(* Offers parameters for SB method (a simple blob detector with multiple thresholds). *)
	{attribute 'TcIecLibraryType'}
{attribute 'Namespace' := 'Tc3_Vision'}
TYPE TcVnParamsSB : 
	STRUCT
		(* Enable filtering by area (fMinArea <= area < fMaxArea). *)
		bFilterByArea : BOOL := TRUE;
		(* Enable filtering by circularity (fMinCircularity <= circularity(4pi * area / perimeter^2) < fMaxCircularity). *)
		bFilterByCircularity : BOOL := FALSE;
		(* Enable filtering by color (thresholdedColor(0 or 255) = nBlobColor). *)
		bFilterByColor : BOOL := FALSE;
		(* Enable filtering by convexity (fMinConvexity <= convexity(area / hullArea) < fMaxConvexity). *)
		bFilterByConvexity : BOOL := FALSE;
		(* Enable filtering by inertia ratio (fMinInertiaRatio <= inertia ratio < fMaxInertiaRatio). *)
		bFilterByInertia : BOOL := FALSE;
		 {attribute 'hide'}
		_reserved1 : ARRAY [1..3] OF USINT;
		(* Min estimated blob area in pixel *)
		fMinArea : REAL := 25;
		(* Max estimated blob area in pixel *)
		fMaxArea : REAL := 15000;
		(* Min circularity (1.0: ideal circle, < 1: less circular, 0: not circular at all) *)
		fMinCircularity : REAL := 0;
		(* Max circularity (1.0: ideal circle, < 1: less circular, 0: not circular at all) *)
		fMaxCircularity : REAL := 1;
		(* 0 or 255 *)
		nBlobColor : USINT := 255;
		 {attribute 'hide'}
		_reserved2 : ARRAY [1..3] OF USINT;
		(* Min convexity (1.0: blob fully convex, < 1: less convex) *)
		fMinConvexity : REAL := 0;
		(* Max convexity (1.0: blob fully convex, < 1: less convex) *)
		fMaxConvexity : REAL := 1;
		(* Min inertia ratio (0.0 .. 1.0) *)
		fMinInertiaRatio : REAL := 0;
		(* Max inertia ratio (0.0 .. 1.0) *)
		fMaxInertiaRatio : REAL := 1;
		(* Min distance between different blobs *)
		fMinBlobDist : REAL := 5;
		(* Min number of same detected blobs (dist < fMinBlobDist) in different thresholds *)
		nMinRepeatability : UDINT := 2;
		(* Min threshold (start) *)
		fMinThreshold : REAL := 30;
		(* Max threshold (stop) *)
		fMaxThreshold : REAL := 225;
		(* Threshold step between min and max threshold *)
		fThresholdStep : REAL := 10;
	END_STRUCT
END_TYPE

// TC_IID_LIST

VAR_GLOBAL
	// Interface ID for interface ITcVnCustomContainerOperation_ITcVnContainer
	{attribute 'tc_no_symbol'}
	IID_ITcVnCustomContainerOperation_ITcVnContainer: IID := (Data1 := 16#6F849123, Data2 := 16#F0E5, Data3 := 16#4EF8, Data4 := [16#99, 16#AF, 16#94, 16#C8, 16#96, 16#DC, 16#45, 16#CA]);
	// Interface ID for interface ITcVnCustomContainerOperation_ITcVnForwardIterator
	{attribute 'tc_no_symbol'}
	IID_ITcVnCustomContainerOperation_ITcVnForwardIterator: IID := (Data1 := 16#49CDB7B5, Data2 := 16#1479, Data3 := 16#4673, Data4 := [16#87, 16#51, 16#92, 16#33, 16#78, 16#F3, 16#BF, 16#4C]);
	// Interface ID for interface ITcVnCustomElementCondition_ITcVnContainer
	{attribute 'tc_no_symbol'}
	IID_ITcVnCustomElementCondition_ITcVnContainer: IID := (Data1 := 16#6B67C104, Data2 := 16#65D1, Data3 := 16#42AF, Data4 := [16#85, 16#B2, 16#AA, 16#CE, 16#B2, 16#0F, 16#60, 16#47]);
	// Interface ID for interface ITcVnCustomElementCondition_ITcVnForwardIterator
	{attribute 'tc_no_symbol'}
	IID_ITcVnCustomElementCondition_ITcVnForwardIterator: IID := (Data1 := 16#DEAD4E4B, Data2 := 16#9BBF, Data3 := 16#4E69, Data4 := [16#A4, 16#7F, 16#D5, 16#7A, 16#42, 16#C7, 16#39, 16#BC]);
	// Interface ID for interface ITcVnColorModel
	{attribute 'tc_no_symbol'}
	IID_ITcVnColorModel: IID := (Data1 := 16#0C43B589, Data2 := 16#90E8, Data3 := 16#4794, Data4 := [16#90, 16#7B, 16#98, 16#AA, 16#35, 16#28, 16#86, 16#D5]);
END_VAR

// Version/Global_Version
{attribute 'TcGenerated'}
// This function has been automatically generated from the project information.
VAR_GLOBAL CONSTANT
	{attribute 'const_non_replaced'}
	{attribute 'linkalways'}
	stLibVersion_Tc3_Vision : ST_LibVersion := (iMajor := 4, iMinor := 0, iBuild := 1, iRevision := 0, sVersion := '4.0.1.0');
	{attribute 'const_non_replaced'}
	{attribute 'linkalways'}
	sLibraryId_Tc3_Vision : String := 'Beckhoff Automation GmbH|Tc3_Vision|4.0.1.0';
END_VAR

// Global Variables/Global_Variables

	VAR_GLOBAL
		VISION_ADS_TIMEOUT	:	TIME := TIME#5s;	(* Default ADS timeout. *)
	END_VAR

// Function Blocks/Image Acquisition/FB_VN_GevCameraControl

	{attribute 'c++_compatible'}
	{attribute 'external_name' := 'FB_VN_GevCameraControl_GUID_2DB65B36_E37A_57E7_6402_AF0E8419D40D'}
	{attribute 'TcIecLibraryType'}
	(* This FB provides the basic functionality to control a GigE Vision camera and access its calibration data. *)
	FUNCTION_BLOCK FB_VN_GevCameraControl
	VAR
		(* Internal reference to the corresponding TcVnGevImageProvider TcCOM module ID, which needs to be set via TC init symbol. *)
		{attribute 'TcInitSymbol'}
		{attribute 'TcCategoryOID' := 'TcVnGevImageProvider'}
		 {attribute 'GUID' := '18071995-0000-0000-0000-00000000000F'}
		oidITcVnGevImageProvider : OTCID;
		 {attribute 'hide'}
		_reserved1 : UINT_0_32;
		(* Internal stuff *)
		{attribute 'hide'}
		 {attribute 'GUID' := '18071995-0000-0000-0000-000000000018'}
		pInternal : PVOID;
	END_VAR


	(* Delete all images contained in the TcVnGevImageProvider TcCOM module receive queue and reset the corresponding omitted images counter. *)
	METHOD ClearImageQueue : HRESULT
END_METHOD


	(* Close the control channel to the camera. *)
	METHOD CloseCamera : HRESULT
END_METHOD


	(* Internal method *)
	{attribute 'hide'}
	METHOD FB_exit : BOOL
	VAR_INPUT
		(*  if TRUE, the exit method is called for exiting an instance that is copied afterwards (online change). *)
		bInCopyCode : BOOL;
	END_VAR
END_METHOD


	(* Internal method *)
	{attribute 'hide'}
	METHOD FB_init : BOOL
	VAR_INPUT
		(*  if TRUE, the retain variables are initialized (warm start / cold start) *)
		bInitRetains : BOOL;
		(*  if TRUE, the instance afterwards gets moved into the copy code (online change) *)
		bInCopyCode : BOOL;
	END_VAR
END_METHOD


	(* Gets the reference calibration pattern points from the TcVnGevImageProvider TcCOM module (Can be set from the calibration assistant) *)
	METHOD GetCalibPatternRef : HRESULT
	VAR_INPUT
		(* Returns the reference calibration pattern points (ContainerType_Vector_TcVnPoint3_REAL) *)
 {attribute 'GUID' := 'BC72B333-E095-465B-9693-7979773CA3B8'}
				ipCalibPatternRef : REFERENCE TO ITcVnContainer;
	END_VAR
END_METHOD


	(* Gets the camera matrix from the TcVnGevImageProvider TcCOM module (requires intrinsic calibration parameters, e.g. set by the calibration assistant) *)
	METHOD GetCameraMatrix : HRESULT
	VAR_INPUT
		(* Returns the camera matrix *)
 {attribute 'GUID' := '91A420A3-4727-4481-B3BB-170528E5BC7C'}
		 {attribute 'Namespace' := 'VN'}
				aCameraMatrix : REFERENCE TO TcVnMatrix3x3_LREAL;
	END_VAR
END_METHOD


	(* Gets the current available image (first in receive queue). *)
	METHOD GetCurrentImage : HRESULT
	VAR_INPUT
		(* Returns the image *)
 {attribute 'GUID' := '70D42C6D-6F4E-4719-8B29-2883D5D59B1C'}
				ipImage : REFERENCE TO ITcVnImage;
	END_VAR
END_METHOD


	(* Gets the current available image (first in receive queue) with undistortion applied (requires intrinsic calibration parameters in the TcVnGevImageProvider TcCOM module, e.g. set by the calibration assistant) *)
	METHOD GetCurrentImageUndistorted : HRESULT
	VAR_INPUT
		(* Returns the undistorted image *)
 {attribute 'GUID' := '70D42C6D-6F4E-4719-8B29-2883D5D59B1C'}
				ipImage : REFERENCE TO ITcVnImage;
	END_VAR
END_METHOD


	(* Gets the current available image (first in receive queue) and its corresponding GVSP info. *)
	METHOD GetCurrentImageWithGvspInfo : HRESULT
	VAR_INPUT
		(* Returns the image *)
 {attribute 'GUID' := '70D42C6D-6F4E-4719-8B29-2883D5D59B1C'}
				ipImage : REFERENCE TO ITcVnImage;
		(* Returns the GVSP info *)
 {attribute 'GUID' := '63FC7E33-91CD-44CD-9015-0BD1DC25722C'}
				stGvspInfo : REFERENCE TO GVSP_IMAGE_INFO;
	END_VAR
END_METHOD


	(* Gets the current available image (first in receive queue) with its corresponding GVSP info and undistortion applied (requires intrinsic calibration parameters in the TcVnGevImageProvider TcCOM module, e.g. set by the calibration assistant) *)
	METHOD GetCurrentImageWithGvspInfoUndistorted : HRESULT
	VAR_INPUT
		(* Returns the undistorted image *)
 {attribute 'GUID' := '70D42C6D-6F4E-4719-8B29-2883D5D59B1C'}
				ipImage : REFERENCE TO ITcVnImage;
		(* Returns the GVSP info *)
 {attribute 'GUID' := '63FC7E33-91CD-44CD-9015-0BD1DC25722C'}
				stGvspInfo : REFERENCE TO GVSP_IMAGE_INFO;
	END_VAR
END_METHOD


	(* Gets the distortion coefficients from the TcVnGevImageProvider TcCOM module (requires intrinsic calibration parameters, e.g. set by the calibration assistant) *)
	METHOD GetDistortionCoefficients : HRESULT
	VAR_INPUT
		(* Returns the distortion coefficients [k1, k2, p1, p2, k3, k4, k5, k6] *)
 {attribute 'GUID' := 'DD112102-C23A-4B37-A43A-A96400B57010'}
		 {attribute 'Namespace' := 'VN'}
				aDistortionCoefficients : REFERENCE TO TcVnArray8_LREAL;
	END_VAR
END_METHOD


	(* Gets the last received image from the queue. *)
	METHOD GetLastImageFromQueue : HRESULT
	VAR_INPUT
		(* Returns the image *)
 {attribute 'GUID' := '70D42C6D-6F4E-4719-8B29-2883D5D59B1C'}
				ipImage : REFERENCE TO ITcVnImage;
	END_VAR
END_METHOD


	(* Gets the number of omitted images since the last call of ClearImageQueue(). If the image receive queue in the TcVnGevImageProvider TcCOM module is full and a new image arrives, the first one in the queue will be deleted and the omitted counter is increased. *)
	METHOD GetOmittedImagesNum : HRESULT
	VAR_INPUT
		(* Returns the number of omitted images *)
		nOmitted : REFERENCE TO ULINT;
	END_VAR
END_METHOD


	(* Gets the rotation matrix from the TcVnGevImageProvider TcCOM module (requires extrinsic calibration parameters, e.g. set by the calibration assistant) *)
	METHOD GetRotationMatrix : HRESULT
	VAR_INPUT
		(* Returns the rotation matrix *)
 {attribute 'GUID' := '91A420A3-4727-4481-B3BB-170528E5BC7C'}
		 {attribute 'Namespace' := 'VN'}
				aRotationMatrix : REFERENCE TO TcVnMatrix3x3_LREAL;
	END_VAR
END_METHOD


	(* Gets the current state of the internal camera control state machine. *)
	METHOD GetState : ETcVnCameraState
END_METHOD


	(* Gets the translation vector from the TcVnGevImageProvider TcCOM module (requires extrinsic calibration parameters, e.g. set by the calibration assistant) *)
	METHOD GetTranslationVector : HRESULT
	VAR_INPUT
		(* Returns the translation vector *)
 {attribute 'GUID' := 'B9A67DEB-A7D1-4F25-95A3-4A82FA5C1E28'}
		 {attribute 'Namespace' := 'VN'}
				aTranslationVector : REFERENCE TO TcVnVector3_LREAL;
	END_VAR
END_METHOD


	(* Initialize the camera to the intended state (includes sending the 'InitCameraCommands' defined in the GevImageAcquisition TcCOM module to the camera). *)
	METHOD InitializeCamera : HRESULT
END_METHOD


	(* Open a control channel to the camera. *)
	METHOD OpenCamera : HRESULT
END_METHOD


	(* Reset the camera controller to initial state (might require multiple calls depending on current state, until S_OK is returned) *)
	METHOD Reset : HRESULT
END_METHOD


	(* Reset the camera features to initial state (sends the 'InitCameraCommands' defined in the GevImageAcquisition TcCOM module to the camera). *)
	METHOD ResetCameraFeatures : HRESULT
END_METHOD


	(* Sets the camera matrix to the TcVnGevImageProvider TcCOM module *)
	METHOD SetCameraMatrix : HRESULT
	VAR_INPUT
		(* The camera matrix to be copied to the TcCOM module *)
 {attribute 'GUID' := '91A420A3-4727-4481-B3BB-170528E5BC7C'}
		 {attribute 'Namespace' := 'VN'}
				aCameraMatrix : REFERENCE TO TcVnMatrix3x3_LREAL;
	END_VAR
END_METHOD


	(* Sets the distortion coefficients to the TcVnGevImageProvider TcCOM module *)
	METHOD SetDistortionCoefficients : HRESULT
	VAR_INPUT
		(* The distortion coefficients to be copied to the TcCOM module *)
 {attribute 'GUID' := 'DD112102-C23A-4B37-A43A-A96400B57010'}
		 {attribute 'Namespace' := 'VN'}
				aDistortionCoefficients : REFERENCE TO TcVnArray8_LREAL;
	END_VAR
END_METHOD


	(* Sets the rotation matrix to the TcVnGevImageProvider TcCOM module *)
	METHOD SetRotationMatrix : HRESULT
	VAR_INPUT
		(* The rotation matrix to be copied to the TcCOM module *)
 {attribute 'GUID' := '91A420A3-4727-4481-B3BB-170528E5BC7C'}
		 {attribute 'Namespace' := 'VN'}
				aRotationMatrix : REFERENCE TO TcVnMatrix3x3_LREAL;
	END_VAR
END_METHOD


	(* Sets the translation vector to the TcVnGevImageProvider TcCOM module *)
	METHOD SetTranslationVector : HRESULT
	VAR_INPUT
		(* The translation vector to be copied to the TcCOM module *)
 {attribute 'GUID' := 'B9A67DEB-A7D1-4F25-95A3-4A82FA5C1E28'}
		 {attribute 'Namespace' := 'VN'}
				aTranslationVector : REFERENCE TO TcVnVector3_LREAL;
	END_VAR
END_METHOD


	(* Send the 'StartAcquisitionCommands' defined in the TcVnGevImageProvider TcCOM module to the camera. *)
	METHOD StartAcquisition : HRESULT
END_METHOD


	(* Send the 'StopAcquisitionCommands' defined in the TcVnGevImageProvider TcCOM module to the camera. *)
	METHOD StopAcquisition : HRESULT
END_METHOD


	(* Send the 'SoftwareTriggerCommands' defined in the TcVnGevImageProvider TcCOM module to the camera. *)
	METHOD TriggerImage : HRESULT
END_METHOD

END_FUNCTION_BLOCK

// Function Blocks/Image Acquisition/FB_VN_FileSourceControl

	{attribute 'c++_compatible'}
	{attribute 'external_name' := 'FB_VN_FileSourceControl_GUID_D3461ABD_28B4_5B2E_777A_A26F58BA9E79'}
	{attribute 'TcIecLibraryType'}
	(* This FB provides access to the images send by a File SOurce instance. *)
	FUNCTION_BLOCK FB_VN_FileSourceControl
	VAR
		(* Internal reference to the corresponding TcVnFileImageProvider TcCOM module ID, which needs to be set via TC init symbol. *)
		{attribute 'TcInitSymbol'}
		{attribute 'TcCategoryOID' := 'TcVnFileImageProvider'}
		 {attribute 'GUID' := '18071995-0000-0000-0000-00000000000F'}
		oidITcVnFileImageProvider : OTCID;
		 {attribute 'hide'}
		_reserved1 : UINT_0_32;
		(* Internal reference to private data. *)
		{attribute 'hide'}
		 {attribute 'GUID' := '18071995-0000-0000-0000-000000000018'}
		pPriv : PVOID;
	END_VAR


	(* Internal method *)
	{attribute 'hide'}
	METHOD FB_exit : BOOL
	VAR_INPUT
		(* If TRUE, the exit method is called for exiting an instance that is copied afterwards (online change). *)
		bInCopyCode : BOOL;
	END_VAR
END_METHOD


	(* Internal method *)
	{attribute 'hide'}
	METHOD FB_init : BOOL
	VAR_INPUT
		(* If TRUE, the retain variables are initialized (warm start / cold start) *)
		bInitRetains : BOOL;
		(* If TRUE, the exit method is called for exiting an instance that is copied afterwards (online change). *)
		bInCopyCode : BOOL;
	END_VAR
END_METHOD


	(* Gets the current available image (if any). *)
	METHOD GetCurrentImage : HRESULT
	VAR_INPUT
		(* Returns the image *)
 {attribute 'GUID' := '70D42C6D-6F4E-4719-8B29-2883D5D59B1C'}
				ipImage : REFERENCE TO ITcVnImage;
	END_VAR
END_METHOD


	(* Gets the current available image (if any) and the corresponding file name. *)
	METHOD GetCurrentImageAndFileName : HRESULT
	VAR_INPUT
		(* Returns the image *)
 {attribute 'GUID' := '70D42C6D-6F4E-4719-8B29-2883D5D59B1C'}
				ipImage : REFERENCE TO ITcVnImage;
	END_VAR
	VAR_IN_OUT CONSTANT
		(* Returns the file name *)
 {attribute 'GUID' := '18071995-0000-0000-0000-00000000001A'}
				sFileName : STRING;
	END_VAR
	VAR_INPUT
		(* Define the maximum allowed length for the file name *)
		nMaxLen : UINT;
	END_VAR
END_METHOD


	(* Activates the File Source. If not in trigger mode, it will start sending images. *)
	METHOD StartAcquisition : HRESULT
END_METHOD


	(* Deactivates the File Source. It will stop sending images. *)
	METHOD StopAcquisition : HRESULT
END_METHOD


	(* Reset the controller to initial state (might require multiple calls depending on current state, until S_OK is returned) *)
	METHOD Reset : HRESULT
END_METHOD


	(* Gets the current state of the internal camera control state machine. *)
	METHOD GetState : ETcVnCameraState
END_METHOD


	(* If in trigger mode, this function triggers the next image in the list. *)
	METHOD TriggerImage : HRESULT
END_METHOD


	(* If in trigger mode, this function triggers a specific image in the list. *)
	METHOD TriggerImageExp : HRESULT
	VAR_INPUT
		(* Amount of images to skip, relative to current *)
		nSkipImages : DINT;
	END_VAR
END_METHOD


	(* If in trigger mode, this function triggers a specific image in the list by name. *)
	METHOD TriggerImageByName : HRESULT
	VAR_IN_OUT CONSTANT
		(* Name of the image to trigger *)
 {attribute 'GUID' := '18071995-0000-0000-0000-00000000001A'}
				sImageName : STRING;
	END_VAR
END_METHOD

END_FUNCTION_BLOCK

// Function Blocks/Image Acquisition/FB_VN_SimpleCameraControl

	{attribute 'c++_compatible'}
	{attribute 'external_name' := 'FB_VN_SimpleCameraControl_GUID_596884A6_7939_51BE_6474_E09301FABEF5'}
	{attribute 'TcIecLibraryType'}
	(* This FB provides the basic functionality to control a camera or a FileSource. *)
	FUNCTION_BLOCK FB_VN_SimpleCameraControl
	VAR
		(* Internal reference to the corresponding TcVnImageProvider TcCOM module ID, which needs to be set via TC init symbol. *)
		{attribute 'TcInitSymbol'}
		{attribute 'TcCategoryOID' := 'TcVnImageProvider'}
		 {attribute 'GUID' := '18071995-0000-0000-0000-00000000000F'}
		oidITcVnImageProvider : OTCID;
		 {attribute 'hide'}
		_reserved1 : UINT_0_32;
		(* Internal stuff *)
		{attribute 'hide'}
		 {attribute 'GUID' := '18071995-0000-0000-0000-000000000018'}
		pInternal : PVOID;
	END_VAR


	(* Internal method *)
	{attribute 'hide'}
	METHOD FB_exit : BOOL
	VAR_INPUT
		(*  if TRUE, the exit method is called for exiting an instance that is copied afterwards (online change). *)
		bInCopyCode : BOOL;
	END_VAR
END_METHOD


	(* Internal method *)
	{attribute 'hide'}
	METHOD FB_init : BOOL
	VAR_INPUT
		(*  if TRUE, the retain variables are initialized (warm start / cold start) *)
		bInitRetains : BOOL;
		(*  if TRUE, the instance afterwards gets moved into the copy code (online change) *)
		bInCopyCode : BOOL;
	END_VAR
END_METHOD


	(* Get the current available image (if any). *)
	METHOD GetCurrentImage : HRESULT
	VAR_INPUT
		(* Returns the image *)
 {attribute 'GUID' := '70D42C6D-6F4E-4719-8B29-2883D5D59B1C'}
				ipImage : REFERENCE TO ITcVnImage;
	END_VAR
END_METHOD


	(* Get the current state of the internal camera control state machine. *)
	METHOD GetState : ETcVnCameraState
END_METHOD


	(* Reset the camera to initial state (might require multiple calls depending on current state, until S_OK is returned) *)
	METHOD Reset : HRESULT
END_METHOD


	(* Start the image acquisition. *)
	METHOD StartAcquisition : HRESULT
END_METHOD


	(* Stop the image acquisition. *)
	METHOD StopAcquisition : HRESULT
END_METHOD


	(* Trigger the next image. *)
	METHOD TriggerImage : HRESULT
END_METHOD

END_FUNCTION_BLOCK

// Function Blocks/File Access/FB_VN_ReadCalibrationPattern

	{attribute 'c++_compatible'}
	{attribute 'external_name' := 'FB_VN_ReadCalibrationPattern_GUID_6F6C0285_AE36_593E_715F_1179FEF2DFE8'}
	{attribute 'TcIecLibraryType'}
	(* This FB reads calibration pattern reference points from an xml file on the targte pc. *)
	FUNCTION_BLOCK FB_VN_ReadCalibrationPattern
	VAR_IN_OUT CONSTANT
		(* Full path of the file or relative path to the default directory on the target pc (%TWINCAT3DIR%\\CustomConfig\\Vision\\CalibrationPattern) *)
		 {attribute 'GUID' := '18071995-0000-0000-0000-00000000001A'}
		sFilePath : STRING;
	END_VAR
	VAR_INPUT
		(* Returns a container with the pattern points (ContainerType_Vector_TcVnPoint3_REAL) *)
		 {attribute 'GUID' := 'BC72B333-E095-465B-9693-7979773CA3B8'}
		ipDestContainer : REFERENCE TO ITcVnContainer;
		(* Reading the file is triggered by a rising edge at this input. *)
		bRead : BOOL;
	END_VAR
	VAR
		 {attribute 'hide'}
		_reserved1 : ARRAY [1..3] OF USINT;
	END_VAR
	VAR_INPUT
		(* Indicates the time before the function is cancelled. *)
		nTimeout : TIME := VISION_ADS_TIMEOUT;
	END_VAR
	VAR_OUTPUT
		(* This output remains TRUE until the function block has executed a command, but at the longest for the duration supplied to the 'nTimeout' input. While bBusy = TRUE, no new command will be accepted at the inputs. *)
		bBusy : BOOL;
		(* This output is switched to TRUE as soon as an error occurs during the execution of a command. The command-specific error code is contained in ‘nErrorId’. If the function block has a timeout error, 'bError' is TRUE and 'nErrorId' is 1861 (hexadecimal 0x745). Is reset to FALSE by the execution of a command at the inputs. *)
		bError : BOOL;
	END_VAR
	VAR
		 {attribute 'hide'}
		_reserved2 : UINT;
	END_VAR
	VAR_OUTPUT
		(* Contains the ADS error code or the command-specific error code of the last executed command. Is reset to 0 by the execution of a command at the inputs. *)
		nErrorId : UDINT;
	END_VAR
	VAR
		(* Internal parameter *)
		{attribute 'hide'}
		nAdsInvStamp : UINT;
		(* Internal parameter *)
		{attribute 'hide'}
		nAdsInvCnt : BYTE;
		(* Internal parameter *)
		{attribute 'hide'}
		ePendingRequest : BYTE;
		(* Internal parameter *)
		{attribute 'hide'}
		nTimeElapsed : TIME;
		(* Internal parameter *)
		{attribute 'hide'}
		bLastRead : BOOL;
		 {attribute 'hide'}
		_reserved3 : UINT_24_56;
		(* Internal parameter *)
		{attribute 'hide'}
		 {attribute 'GUID' := '18071995-0000-0000-0000-000000000018'}
		pBuffer : PVOID;
	END_VAR


	(* Internal method *)
	{attribute 'hide'}
	METHOD FB_exit : BOOL
	VAR_INPUT
		(*  if TRUE, the exit method is called for exiting an instance that is copied afterwards (online change). *)
		bInCopyCode : BOOL;
	END_VAR
END_METHOD


	(* Internal method *)
	{attribute 'hide'}
	METHOD FB_init : BOOL
	VAR_INPUT
		(*  if TRUE, the retain variables are initialized (warm start / cold start) *)
		bInitRetains : BOOL;
		(*  if TRUE, the instance afterwards gets moved into the copy code (online change) *)
		bInCopyCode : BOOL;
	END_VAR
END_METHOD

END_FUNCTION_BLOCK

// Function Blocks/File Access/FB_VN_ReadContainer

	{attribute 'c++_compatible'}
	{attribute 'external_name' := 'FB_VN_ReadContainer_GUID_95BC104A_73B3_5998_484A_2F368A46664B'}
	{attribute 'TcIecLibraryType'}
	(* This FB reads a container from an xml file on the target pc. *)
	FUNCTION_BLOCK FB_VN_ReadContainer
	VAR_IN_OUT CONSTANT
		(* Full path of the file or relative path to the default directory on the target pc *)
		 {attribute 'GUID' := '18071995-0000-0000-0000-00000000001A'}
		sFilePath : STRING;
	END_VAR
	VAR_INPUT
		(* Returns a container with the loaded content *)
		 {attribute 'GUID' := 'BC72B333-E095-465B-9693-7979773CA3B8'}
		ipDestContainer : REFERENCE TO ITcVnContainer;
		(* The type id of the container to return. If this parameter is not set, a suitable container type will be determined automatically. *)
		 {attribute 'GUID' := '18071995-0000-0000-0000-000000000021'}
		nDestTypeGuid : GUID;
		(* Reading the file is triggered by a rising edge at this input. *)
		bRead : BOOL;
	END_VAR
	VAR
		 {attribute 'hide'}
		_reserved1 : ARRAY [1..3] OF USINT;
	END_VAR
	VAR_INPUT
		(* Indicates the time before the function is cancelled. *)
		nTimeout : TIME := VISION_ADS_TIMEOUT;
	END_VAR
	VAR_OUTPUT
		(* This output remains TRUE until the function block has executed a command, but at the longest for the duration supplied to the 'nTimeout' input. While bBusy = TRUE, no new command will be accepted at the inputs. *)
		bBusy : BOOL;
		(* This output is switched to TRUE as soon as an error occurs during the execution of a command. The command-specific error code is contained in ‘nErrorId’. If the function block has a timeout error, 'bError' is TRUE and 'nErrorId' is 1861 (hexadecimal 0x745). Is reset to FALSE by the execution of a command at the inputs. *)
		bError : BOOL;
	END_VAR
	VAR
		 {attribute 'hide'}
		_reserved2 : UINT;
	END_VAR
	VAR_OUTPUT
		(* Contains the ADS error code or the command-specific error code of the last executed command. Is reset to 0 by the execution of a command at the inputs. *)
		nErrorId : UDINT;
	END_VAR
	VAR
		(* Internal parameter *)
		{attribute 'hide'}
		nAdsInvStamp : UINT;
		(* Internal parameter *)
		{attribute 'hide'}
		nAdsInvCnt : BYTE;
		(* Internal parameter *)
		{attribute 'hide'}
		ePendingRequest : BYTE;
		(* Internal parameter *)
		{attribute 'hide'}
		nTimeElapsed : TIME;
		(* Internal parameter *)
		{attribute 'hide'}
		bLastRead : BOOL;
		 {attribute 'hide'}
		_reserved3 : UINT_24_56;
		(* Internal parameter *)
		{attribute 'hide'}
		 {attribute 'GUID' := '18071995-0000-0000-0000-000000000018'}
		pBuffer : PVOID;
	END_VAR


	(* Internal method *)
	{attribute 'hide'}
	METHOD FB_exit : BOOL
	VAR_INPUT
		(*  if TRUE, the exit method is called for exiting an instance that is copied afterwards (online change). *)
		bInCopyCode : BOOL;
	END_VAR
END_METHOD


	(* Internal method *)
	{attribute 'hide'}
	METHOD FB_init : BOOL
	VAR_INPUT
		(*  if TRUE, the retain variables are initialized (warm start / cold start) *)
		bInitRetains : BOOL;
		(*  if TRUE, the instance afterwards gets moved into the copy code (online change) *)
		bInCopyCode : BOOL;
	END_VAR
END_METHOD

END_FUNCTION_BLOCK

// Function Blocks/File Access/FB_VN_ReadImage

	{attribute 'c++_compatible'}
	{attribute 'external_name' := 'FB_VN_ReadImage_GUID_00EE7AEB_0E5B_5975_559A_9672FFADF570'}
	{attribute 'TcIecLibraryType'}
	(* This FB reads an image from a file on the target pc. *)
	FUNCTION_BLOCK FB_VN_ReadImage
	VAR_IN_OUT CONSTANT
		(* Full path of the file or relative path to the default image directory on the target pc *)
		 {attribute 'GUID' := '18071995-0000-0000-0000-00000000001A'}
		sFilePath : STRING;
	END_VAR
	VAR_INPUT
		(* Returns an image with the loaded content *)
		 {attribute 'GUID' := '70D42C6D-6F4E-4719-8B29-2883D5D59B1C'}
		ipDestImage : REFERENCE TO ITcVnImage;
		(* Reading the file is triggered by a rising edge at this input. *)
		bRead : BOOL;
	END_VAR
	VAR
		 {attribute 'hide'}
		_reserved1 : ARRAY [1..3] OF USINT;
	END_VAR
	VAR_INPUT
		(* Indicates the time before the function is cancelled. *)
		nTimeout : TIME := VISION_ADS_TIMEOUT;
	END_VAR
	VAR_OUTPUT
		(* This output remains TRUE until the function block has executed a command, but at the longest for the duration supplied to the 'nTimeout' input. While bBusy = TRUE, no new command will be accepted at the inputs. *)
		bBusy : BOOL;
		(* This output is switched to TRUE as soon as an error occurs during the execution of a command. The command-specific error code is contained in ‘nErrorId’. If the function block has a timeout error, 'bError' is TRUE and 'nErrorId' is 1861 (hexadecimal 0x745). Is reset to FALSE by the execution of a command at the inputs. *)
		bError : BOOL;
	END_VAR
	VAR
		 {attribute 'hide'}
		_reserved2 : UINT;
	END_VAR
	VAR_OUTPUT
		(* Contains the ADS error code or the command-specific error code of the last executed command. Is reset to 0 by the execution of a command at the inputs. *)
		nErrorId : UDINT;
	END_VAR
	VAR
		(* Internal parameter *)
		{attribute 'hide'}
		nAdsInvStamp : UINT;
		(* Internal parameter *)
		{attribute 'hide'}
		nAdsInvCnt : BYTE;
		(* Internal parameter *)
		{attribute 'hide'}
		ePendingRequest : BYTE;
		(* Internal parameter *)
		{attribute 'hide'}
		nTimeElapsed : TIME;
		(* Internal parameter *)
		{attribute 'hide'}
		bLastRead : BOOL;
		 {attribute 'hide'}
		_reserved3 : UINT_24_56;
		(* Internal parameter *)
		{attribute 'hide'}
		 {attribute 'GUID' := '18071995-0000-0000-0000-000000000018'}
		pBuffer : PVOID;
	END_VAR


	(* Internal method *)
	{attribute 'hide'}
	METHOD FB_exit : BOOL
	VAR_INPUT
		(*  if TRUE, the exit method is called for exiting an instance that is copied afterwards (online change). *)
		bInCopyCode : BOOL;
	END_VAR
END_METHOD


	(* Internal method *)
	{attribute 'hide'}
	METHOD FB_init : BOOL
	VAR_INPUT
		(*  if TRUE, the retain variables are initialized (warm start / cold start) *)
		bInitRetains : BOOL;
		(*  if TRUE, the instance afterwards gets moved into the copy code (online change) *)
		bInCopyCode : BOOL;
	END_VAR
END_METHOD

END_FUNCTION_BLOCK

// Function Blocks/File Access/FB_VN_WriteContainer

	{attribute 'c++_compatible'}
	{attribute 'external_name' := 'FB_VN_WriteContainer_GUID_A59DFE63_73F8_599A_4B41_282C9273F4F7'}
	{attribute 'TcIecLibraryType'}
	(* This FB writes a container as an xml file to the hard drive. *)
	FUNCTION_BLOCK FB_VN_WriteContainer
	VAR_INPUT
		(* The container to write *)
		 {attribute 'GUID' := 'BC72B333-E095-465B-9693-7979773CA3B8'}
		ipContainer : REFERENCE TO ITcVnContainer;
	END_VAR
	VAR_IN_OUT CONSTANT
		(* Full path of the file or relative path to the default directory on the target pc (e.g. only a file name). If the string is empty, a file name will be generated (containing the current time). *)
		 {attribute 'GUID' := '18071995-0000-0000-0000-00000000001A'}
		sFilePath : STRING;
	END_VAR
	VAR_INPUT
		(* Container export format (default is human readable xml) *)
		 {attribute 'GUID' := 'F8305D79-70A3-4F93-A939-2FF3B8D6AF74'}
		 {attribute 'Namespace' := 'Tc3_Vision'}
		eExportFormat : ETcVnContainerExportFormat := TCVN_CEF_XML;
		(* Writing the container is triggered by a rising edge at this input. *)
		bWrite : BOOL;
	END_VAR
	VAR
		 {attribute 'hide'}
		_reserved1 : USINT;
	END_VAR
	VAR_INPUT
		(* Indicates the time before the function is cancelled. *)
		nTimeout : TIME := VISION_ADS_TIMEOUT;
	END_VAR
	VAR_OUTPUT
		(* This output remains TRUE until the function block has executed a command, but at the longest for the duration supplied to the 'nTimeout' input. While bBusy = TRUE, no new command will be accepted at the inputs. *)
		bBusy : BOOL;
		(* This output is switched to TRUE as soon as an error occurs during the execution of a command. The command-specific error code is contained in ‘nErrorId’. If the function block has a timeout error, 'bError' is TRUE and 'nErrorId' is 1861 (hexadecimal 0x745). Is reset to FALSE by the execution of a command at the inputs. *)
		bError : BOOL;
	END_VAR
	VAR
		 {attribute 'hide'}
		_reserved2 : UINT;
	END_VAR
	VAR_OUTPUT
		(* Contains the ADS error code or the command-specific error code of the last executed command. Is reset to 0 by the execution of a command at the inputs. *)
		nErrorId : UDINT;
	END_VAR
	VAR
		(* Internal parameter *)
		{attribute 'hide'}
		nAdsInvStamp : UINT;
		(* Internal parameter *)
		{attribute 'hide'}
		nAdsInvCnt : BYTE;
		 {attribute 'hide'}
		_reserved3 : USINT;
		(* Internal parameter *)
		{attribute 'hide'}
		nTimeElapsed : TIME;
		(* Internal parameter *)
		{attribute 'hide'}
		bLastWrite : BOOL;
		 {attribute 'hide'}
		_reserved4 : UINT_24_56;
	END_VAR


	(* Internal method *)
	{attribute 'hide'}
	METHOD FB_exit : BOOL
	VAR_INPUT
		(* If TRUE, the exit method is called for exiting an instance that is copied afterwards (online change). *)
		bInCopyCode : BOOL;
	END_VAR
END_METHOD


	(* Internal method *)
	{attribute 'hide'}
	METHOD FB_init : BOOL
	VAR_INPUT
		(* If TRUE, the retain variables are initialized (warm start / cold start) *)
		bInitRetains : BOOL;
		(* If TRUE, the instance afterwards gets moved into the copy code (online change) *)
		bInCopyCode : BOOL;
	END_VAR
END_METHOD

END_FUNCTION_BLOCK

// Function Blocks/File Access/FB_VN_WriteImage

	{attribute 'c++_compatible'}
	{attribute 'external_name' := 'FB_VN_WriteImage_GUID_4B9DB54D_E8F3_555D_4A92_9CFCB0664FA2'}
	{attribute 'TcIecLibraryType'}
	(* This FB writes an image to the hard drive. *)
	FUNCTION_BLOCK FB_VN_WriteImage
	VAR_INPUT
		(* The image to write *)
		 {attribute 'GUID' := '70D42C6D-6F4E-4719-8B29-2883D5D59B1C'}
		ipImage : REFERENCE TO ITcVnImage;
	END_VAR
	VAR_IN_OUT CONSTANT
		(* Full path of the file or relative path to the default directory on the target pc (e.g. only a file name). If the string is empty, a file name will be generated (containing the current time). *)
		 {attribute 'GUID' := '18071995-0000-0000-0000-00000000001A'}
		sFilePath : STRING;
	END_VAR
	VAR_INPUT
		(* Writing the image is triggered by a rising edge at this input. *)
		bWrite : BOOL;
	END_VAR
	VAR
		 {attribute 'hide'}
		_reserved1 : ARRAY [1..3] OF USINT;
	END_VAR
	VAR_INPUT
		(* Indicates the time before the function is cancelled. *)
		nTimeout : TIME := VISION_ADS_TIMEOUT;
	END_VAR
	VAR_OUTPUT
		(* This output remains TRUE until the function block has executed a command, but at the longest for the duration supplied to the 'nTimeout' input. While bBusy = TRUE, no new command will be accepted at the inputs. *)
		bBusy : BOOL;
		(* This output is switched to TRUE as soon as an error occurs during the execution of a command. The command-specific error code is contained in ‘nErrorId’. If the function block has a timeout error, 'bError' is TRUE and 'nErrorId' is 1861 (hexadecimal 0x745). Is reset to FALSE by the execution of a command at the inputs. *)
		bError : BOOL;
	END_VAR
	VAR
		 {attribute 'hide'}
		_reserved2 : UINT;
	END_VAR
	VAR_OUTPUT
		(* Contains the ADS error code or the command-specific error code of the last executed command. Is reset to 0 by the execution of a command at the inputs. *)
		nErrorId : UDINT;
	END_VAR
	VAR
		(* Internal parameter *)
		{attribute 'hide'}
		nAdsInvStamp : UINT;
		(* Internal parameter *)
		{attribute 'hide'}
		nAdsInvCnt : BYTE;
		 {attribute 'hide'}
		_reserved3 : USINT;
		(* Internal parameter *)
		{attribute 'hide'}
		nTimeElapsed : TIME;
		(* Internal parameter *)
		{attribute 'hide'}
		bLastWrite : BOOL;
		 {attribute 'hide'}
		_reserved4 : UINT_24_56;
	END_VAR


	(* Internal method *)
	{attribute 'hide'}
	METHOD FB_exit : BOOL
	VAR_INPUT
		(*  if TRUE, the exit method is called for exiting an instance that is copied afterwards (online change). *)
		bInCopyCode : BOOL;
	END_VAR
END_METHOD


	(* Internal method *)
	{attribute 'hide'}
	METHOD FB_init : BOOL
	VAR_INPUT
		(*  if TRUE, the retain variables are initialized (warm start / cold start) *)
		bInitRetains : BOOL;
		(*  if TRUE, the instance afterwards gets moved into the copy code (online change) *)
		bInCopyCode : BOOL;
	END_VAR
END_METHOD

END_FUNCTION_BLOCK

// Function Blocks/Camera Register Access/FB_VN_ReadRegister_UDINT

	{attribute 'c++_compatible'}
	{attribute 'external_name' := 'FB_VN_ReadRegister_UDINT_GUID_5A6880D9_3D24_5A76_5712_175B5A191D07'}
	{attribute 'TcIecLibraryType'}
	(* This FB reads a DINT register from the camera. Requires an open control channel (e.g. by calling FB_VN_GevCameraControl.OpenCamera() before) *)
	FUNCTION_BLOCK FB_VN_ReadRegister_UDINT
	VAR_INPUT
		(* The address of the register that should be read *)
		 {attribute 'GUID' := 'E1ED2436-3512-43FA-B927-3F71DEDDA853'}
		nAddress : GVCP_REGISTER_ADDRESS;
		(* OPTIONAL: The endianness of the register. 0 = Big, 1 = Little. Default: 0 *)
		nEndian : UINT;
		(* Reading the register is triggered by a rising edge at this input. *)
		bRead : BOOL;
	END_VAR
	VAR
		 {attribute 'hide'}
		_reserved1 : USINT;
	END_VAR
	VAR_INPUT
		(* Indicates the time before the function is cancelled. *)
		nTimeout : TIME := VISION_ADS_TIMEOUT;
	END_VAR
	VAR_OUTPUT
		(* The read value *)
		nValue : UDINT;
		(* This output remains TRUE until the function block has executed a command, but at the longest for the duration supplied to the 'nTimeout' input. While bBusy = TRUE, no new command will be accepted at the inputs. *)
		bBusy : BOOL;
		(* This output is switched to TRUE as soon as an error occurs during the execution of a command. The command-specific error code is contained in ‘nErrorId’. If the function block has a timeout error, 'bError' is TRUE and 'nErrorId' is 1861 (hexadecimal 0x745). Is reset to FALSE by the execution of a command at the inputs. *)
		bError : BOOL;
	END_VAR
	VAR
		 {attribute 'hide'}
		_reserved2 : UINT;
	END_VAR
	VAR_OUTPUT
		(* Contains the ADS error code or the command-specific error code of the last executed command. Is reset to 0 by the execution of a command at the inputs. *)
		nErrorId : UDINT;
	END_VAR
	VAR
		(* Internal reference to the corresponding TcVnGevImageProvider TcCOM module ID, which needs to be set via TC init symbol. *)
		{attribute 'TcInitSymbol'}
		{attribute 'TcCategoryOID' := 'TcVnGevImageProvider'}
		 {attribute 'GUID' := '18071995-0000-0000-0000-00000000000F'}
		oidITcVnGevImageProvider : OTCID;
		 {attribute 'hide'}
		_reserved3 : UINT_0_32;
		(* Internal reference to the corresponding TcVnGevImageProvider module. *)
		{attribute 'hide'}
		 {attribute 'GUID' := 'ED7659DB-95DC-4A4A-B62F-02C9870D5E81'}
		ipGevImageProvider : ITcVnGevImageProvider;
		(* Internal timestamp for timeout detection *)
		{attribute 'hide'}
		nTimeElapsed : TIME;
		(* Internal flag for rising edge detection *)
		{attribute 'hide'}
		bLastRead : BOOL;
		 {attribute 'hide'}
		_reserved4 : ARRAY [1..3] OF USINT;
	END_VAR


	(* Internal method *)
	{attribute 'hide'}
	METHOD FB_exit : BOOL
	VAR_INPUT
		(*  if TRUE, the exit method is called for exiting an instance that is copied afterwards (online change). *)
		bInCopyCode : BOOL;
	END_VAR
END_METHOD


	(* Internal method *)
	{attribute 'hide'}
	METHOD FB_init : BOOL
	VAR_INPUT
		(*  if TRUE, the retain variables are initialized (warm start / cold start) *)
		bInitRetains : BOOL;
		(*  if TRUE, the instance afterwards gets moved into the copy code (online change) *)
		bInCopyCode : BOOL;
	END_VAR
END_METHOD

END_FUNCTION_BLOCK

// Function Blocks/Camera Register Access/FB_VN_WriteRegister_UDINT

	{attribute 'c++_compatible'}
	{attribute 'external_name' := 'FB_VN_WriteRegister_UDINT_GUID_4434B241_E667_50D4_49D0_7991F8DDF3A5'}
	{attribute 'TcIecLibraryType'}
	(* This FB writes a DINT value into a register on the camera. Requires an open control channel (e.g. by calling FB_VN_GevCameraControl.OpenCamera() before) *)
	FUNCTION_BLOCK FB_VN_WriteRegister_UDINT
	VAR_INPUT
		(* The address of the register that should be written *)
		 {attribute 'GUID' := 'E1ED2436-3512-43FA-B927-3F71DEDDA853'}
		nAddress : GVCP_REGISTER_ADDRESS;
		(* The value to write *)
		nValue : UDINT;
		(* OPTIONAL: The endianness of the register. 0 = Big, 1 = Little. Default: 0 *)
		nEndian : UINT;
		(* Reading the register is triggered by a rising edge at this input. *)
		bWrite : BOOL;
	END_VAR
	VAR
		 {attribute 'hide'}
		_reserved1 : USINT;
	END_VAR
	VAR_INPUT
		(* Indicates the time before the function is cancelled. *)
		nTimeout : TIME := VISION_ADS_TIMEOUT;
	END_VAR
	VAR_OUTPUT
		(* This output remains TRUE until the function block has executed a command, but at the longest for the duration supplied to the 'nTimeout' input. While bBusy = TRUE, no new command will be accepted at the inputs. *)
		bBusy : BOOL;
		(* This output is switched to TRUE as soon as an error occurs during the execution of a command. The command-specific error code is contained in ‘nErrorId’. If the function block has a timeout error, 'bError' is TRUE and 'nErrorId' is 1861 (hexadecimal 0x745). Is reset to FALSE by the execution of a command at the inputs. *)
		bError : BOOL;
	END_VAR
	VAR
		 {attribute 'hide'}
		_reserved2 : UINT;
	END_VAR
	VAR_OUTPUT
		(* Contains the ADS error code or the command-specific error code of the last executed command. Is reset to 0 by the execution of a command at the inputs. *)
		nErrorId : UDINT;
	END_VAR
	VAR
		(* Internal reference to the corresponding TcVnGevImageProvider TcCOM module ID, which needs to be set via TC init symbol. *)
		{attribute 'TcInitSymbol'}
		{attribute 'TcCategoryOID' := 'TcVnGevImageProvider'}
		 {attribute 'GUID' := '18071995-0000-0000-0000-00000000000F'}
		oidITcVnGevImageProvider : OTCID;
		 {attribute 'hide'}
		_reserved3 : UINT_0_32;
		(* Internal reference to the corresponding TcVnGevImageProvider module. *)
		{attribute 'hide'}
		 {attribute 'GUID' := 'ED7659DB-95DC-4A4A-B62F-02C9870D5E81'}
		ipGevImageProvider : ITcVnGevImageProvider;
		(* Internal timestamp for timeout detection *)
		{attribute 'hide'}
		nTimeElapsed : TIME;
		(* Internal flag for rising edge detection *)
		{attribute 'hide'}
		bLastWrite : BOOL;
		 {attribute 'hide'}
		_reserved4 : ARRAY [1..3] OF USINT;
	END_VAR


	(* Internal method *)
	{attribute 'hide'}
	METHOD FB_exit : BOOL
	VAR_INPUT
		(*  if TRUE, the exit method is called for exiting an instance that is copied afterwards (online change). *)
		bInCopyCode : BOOL;
	END_VAR
END_METHOD


	(* Internal method *)
	{attribute 'hide'}
	METHOD FB_init : BOOL
	VAR_INPUT
		(*  if TRUE, the retain variables are initialized (warm start / cold start) *)
		bInitRetains : BOOL;
		(*  if TRUE, the instance afterwards gets moved into the copy code (online change) *)
		bInCopyCode : BOOL;
	END_VAR
END_METHOD

END_FUNCTION_BLOCK

// Function Blocks/Camera Register Access/FB_VN_ReadMemory

	{attribute 'c++_compatible'}
	{attribute 'external_name' := 'FB_VN_ReadMemory_GUID_771119DB_D184_56D5_6E01_412391084A54'}
	{attribute 'TcIecLibraryType'}
	(* This FB reads consecutive memory locations from the camera. Requires an open control channel (e.g. by calling FB_VN_GevCameraControl.OpenCamera() before) *)
	FUNCTION_BLOCK FB_VN_ReadMemory
	VAR_INPUT
		(* The address of the first byte to read from the camera (must be 32-bit aligned) *)
		 {attribute 'GUID' := 'E1ED2436-3512-43FA-B927-3F71DEDDA853'}
		nAddress : GVCP_REGISTER_ADDRESS;
		(* The number of bytes to read, starting with nAddress (must be a multiple of 4, not more than 536) *)
		nLength : UINT;
	END_VAR
	VAR
		 {attribute 'hide'}
		_reserved1 : UINT;
	END_VAR
	VAR_INPUT
		(* Pointer to the buffer where the read memory content is written to (The buffer must have a size of at least nLength bytes!) *)
		 {attribute 'GUID' := '18071995-0000-0000-0000-000000000018'}
		pBuffer : PVOID;
		(* Reading the memory is triggered by a rising edge at this input. *)
		bRead : BOOL;
	END_VAR
	VAR
		 {attribute 'hide'}
		_reserved2 : ARRAY [1..3] OF USINT;
	END_VAR
	VAR_INPUT
		(* Indicates the time before the function is cancelled. *)
		nTimeout : TIME := VISION_ADS_TIMEOUT;
	END_VAR
	VAR_OUTPUT
		(* This output remains TRUE until the function block has executed a command, but at the longest for the duration supplied to the 'nTimeout' input. While bBusy = TRUE, no new command will be accepted at the inputs. *)
		bBusy : BOOL;
		(* This output is switched to TRUE as soon as an error occurs during the execution of a command. The command-specific error code is contained in ‘nErrorId’. If the function block has a timeout error, 'bError' is TRUE and 'nErrorId' is 1861 (hexadecimal 0x745). Is reset to FALSE by the execution of a command at the inputs. *)
		bError : BOOL;
	END_VAR
	VAR
		 {attribute 'hide'}
		_reserved3 : UINT;
	END_VAR
	VAR_OUTPUT
		(* Contains the ADS error code or the command-specific error code of the last executed command. Is reset to 0 by the execution of a command at the inputs. *)
		nErrorId : UDINT;
	END_VAR
	VAR
		(* Internal reference to the corresponding TcVnGevImageProvider TcCOM module ID, which needs to be set via TC init symbol. *)
		{attribute 'TcInitSymbol'}
		{attribute 'TcCategoryOID' := 'TcVnGevImageProvider'}
		 {attribute 'GUID' := '18071995-0000-0000-0000-00000000000F'}
		oidITcVnGevImageProvider : OTCID;
		 {attribute 'hide'}
		_reserved4 : UINT_0_32;
		(* Internal reference to the corresponding TcVnGevImageProvider module. *)
		{attribute 'hide'}
		 {attribute 'GUID' := 'ED7659DB-95DC-4A4A-B62F-02C9870D5E81'}
		ipGevImageProvider : ITcVnGevImageProvider;
		(* Internal timestamp for timeout detection *)
		{attribute 'hide'}
		nTimeElapsed : TIME;
		(* Internal flag for rising edge detection *)
		{attribute 'hide'}
		bLastRead : BOOL;
		 {attribute 'hide'}
		_reserved5 : ARRAY [1..3] OF USINT;
	END_VAR


	(* Internal method *)
	{attribute 'hide'}
	METHOD FB_exit : BOOL
	VAR_INPUT
		(* If TRUE, the exit method is called for exiting an instance that is copied afterwards (online change). *)
		bInCopyCode : BOOL;
	END_VAR
END_METHOD


	(* Internal method *)
	{attribute 'hide'}
	METHOD FB_init : BOOL
	VAR_INPUT
		(* If TRUE, the retain variables are initialized (warm start / cold start) *)
		bInitRetains : BOOL;
		(* If TRUE, the instance afterwards gets moved into the copy code (online change) *)
		bInCopyCode : BOOL;
	END_VAR
END_METHOD

END_FUNCTION_BLOCK

// Function Blocks/Camera Register Access/FB_VN_WriteMemory

	{attribute 'c++_compatible'}
	{attribute 'external_name' := 'FB_VN_WriteMemory_GUID_62310BC1_989D_5DF1_7D8A_8818DF4CC801'}
	{attribute 'TcIecLibraryType'}
	(* This FB writes data to consecutive memory locations on the camera. Requires an open control channel (e.g. by calling FB_VN_GevCameraControl.OpenCamera() before) *)
	FUNCTION_BLOCK FB_VN_WriteMemory
	VAR_INPUT
		(* The address of the first byte to write to the camera (must be 32-bit aligned) *)
		 {attribute 'GUID' := 'E1ED2436-3512-43FA-B927-3F71DEDDA853'}
		nAddress : GVCP_REGISTER_ADDRESS;
		(* The number of bytes to write, starting at nAddress (must be a multiple of 4, not more than 536) *)
		nLength : UINT;
	END_VAR
	VAR
		 {attribute 'hide'}
		_reserved1 : UINT;
	END_VAR
	VAR_INPUT
		(* Pointer to the data that should be written to the camera (must have a size of at least nLength bytes!) *)
		 {attribute 'GUID' := '18071995-0000-0000-0000-000000000018'}
		pData : PVOID;
		(* Writing the memory is triggered by a rising edge at this input. *)
		bWrite : BOOL;
	END_VAR
	VAR
		 {attribute 'hide'}
		_reserved2 : ARRAY [1..3] OF USINT;
	END_VAR
	VAR_INPUT
		(* Indicates the time before the function is cancelled. *)
		nTimeout : TIME := VISION_ADS_TIMEOUT;
	END_VAR
	VAR_OUTPUT
		(* This output remains TRUE until the function block has executed a command, but at the longest for the duration supplied to the 'nTimeout' input. While bBusy = TRUE, no new command will be accepted at the inputs. *)
		bBusy : BOOL;
		(* This output is switched to TRUE as soon as an error occurs during the execution of a command. The command-specific error code is contained in ‘nErrorId’. If the function block has a timeout error, 'bError' is TRUE and 'nErrorId' is 1861 (hexadecimal 0x745). Is reset to FALSE by the execution of a command at the inputs. *)
		bError : BOOL;
	END_VAR
	VAR
		 {attribute 'hide'}
		_reserved3 : UINT;
	END_VAR
	VAR_OUTPUT
		(* Contains the ADS error code or the command-specific error code of the last executed command. Is reset to 0 by the execution of a command at the inputs. *)
		nErrorId : UDINT;
		(* The number of bytes that have been successfully written to the camera. *)
		nBytesWritten : UINT;
	END_VAR
	VAR
		 {attribute 'hide'}
		_reserved4 : UINT;
		(* Internal reference to the corresponding TcVnGevImageProvider TcCOM module ID, which needs to be set via TC init symbol. *)
		{attribute 'TcInitSymbol'}
		{attribute 'TcCategoryOID' := 'TcVnGevImageProvider'}
		 {attribute 'GUID' := '18071995-0000-0000-0000-00000000000F'}
		oidITcVnGevImageProvider : OTCID;
		(* Internal reference to the corresponding TcVnGevImageProvider module. *)
		{attribute 'hide'}
		 {attribute 'GUID' := 'ED7659DB-95DC-4A4A-B62F-02C9870D5E81'}
		ipGevImageProvider : ITcVnGevImageProvider;
		(* Internal timestamp for timeout detection *)
		{attribute 'hide'}
		nTimeElapsed : TIME;
		(* Internal flag for rising edge detection *)
		{attribute 'hide'}
		bLastRead : BOOL;
		 {attribute 'hide'}
		_reserved5 : ARRAY [1..3] OF USINT;
	END_VAR


	(* Internal method *)
	{attribute 'hide'}
	METHOD FB_exit : BOOL
	VAR_INPUT
		(* If TRUE, the exit method is called for exiting an instance that is copied afterwards (online change). *)
		bInCopyCode : BOOL;
	END_VAR
END_METHOD


	(* Internal method *)
	{attribute 'hide'}
	METHOD FB_init : BOOL
	VAR_INPUT
		(* If TRUE, the retain variables are initialized (warm start / cold start) *)
		bInitRetains : BOOL;
		(* If TRUE, the instance afterwards gets moved into the copy code (online change) *)
		bInCopyCode : BOOL;
	END_VAR
END_METHOD

END_FUNCTION_BLOCK

// Function Blocks/Camera Register Access/FB_VN_ReadRegister_REAL

	{attribute 'c++_compatible'}
	{attribute 'external_name' := 'FB_VN_ReadRegister_REAL_GUID_002B38D5_5613_59B9_615F_491AF89E32A4'}
	{attribute 'TcIecLibraryType'}
	(* This FB reads a REAL register from the camera. Requires an open control channel (e.g. by calling FB_VN_GevCameraControl.OpenCamera() before) *)
	FUNCTION_BLOCK FB_VN_ReadRegister_REAL
	VAR_INPUT
		(* The address of the register that should be read *)
		 {attribute 'GUID' := 'E1ED2436-3512-43FA-B927-3F71DEDDA853'}
		nAddress : GVCP_REGISTER_ADDRESS;
		(* OPTIONAL: The endianness of the register. 0 = Big, 1 = Little. Default: 0 *)
		nEndian : UINT;
		(* Reading the register is triggered by a rising edge at this input. *)
		bRead : BOOL;
	END_VAR
	VAR
		 {attribute 'hide'}
		_reserved1 : USINT;
	END_VAR
	VAR_INPUT
		(* Indicates the time before the function is cancelled. *)
		nTimeout : TIME := VISION_ADS_TIMEOUT;
	END_VAR
	VAR_OUTPUT
		(* The read value *)
		fValue : REAL;
		(* This output remains TRUE until the function block has executed a command, but at the longest for the duration supplied to the 'nTimeout' input. While bBusy = TRUE, no new command will be accepted at the inputs. *)
		bBusy : BOOL;
		(* This output is switched to TRUE as soon as an error occurs during the execution of a command. The command-specific error code is contained in ‘nErrorId’. If the function block has a timeout error, 'bError' is TRUE and 'nErrorId' is 1861 (hexadecimal 0x745). Is reset to FALSE by the execution of a command at the inputs. *)
		bError : BOOL;
	END_VAR
	VAR
		 {attribute 'hide'}
		_reserved2 : UINT;
	END_VAR
	VAR_OUTPUT
		(* Contains the ADS error code or the command-specific error code of the last executed command. Is reset to 0 by the execution of a command at the inputs. *)
		nErrorId : UDINT;
	END_VAR
	VAR
		(* Internal reference to the corresponding TcVnGevImageProvider TcCOM module ID, which needs to be set via TC init symbol. *)
		{attribute 'TcInitSymbol'}
		{attribute 'TcCategoryOID' := 'TcVnGevImageProvider'}
		 {attribute 'GUID' := '18071995-0000-0000-0000-00000000000F'}
		oidITcVnGevImageProvider : OTCID;
		 {attribute 'hide'}
		_reserved3 : UINT_0_32;
		(* Internal reference to the corresponding TcVnGevImageProvider module. *)
		{attribute 'hide'}
		 {attribute 'GUID' := 'ED7659DB-95DC-4A4A-B62F-02C9870D5E81'}
		ipGevImageProvider : ITcVnGevImageProvider;
		(* Internal timestamp for timeout detection *)
		{attribute 'hide'}
		nTimeElapsed : TIME;
		(* Internal flag for rising edge detection *)
		{attribute 'hide'}
		bLastRead : BOOL;
		 {attribute 'hide'}
		_reserved4 : ARRAY [1..3] OF USINT;
	END_VAR


	(* Internal method *)
	{attribute 'hide'}
	METHOD FB_exit : BOOL
	VAR_INPUT
		(*  if TRUE, the exit method is called for exiting an instance that is copied afterwards (online change). *)
		bInCopyCode : BOOL;
	END_VAR
END_METHOD


	(* Internal method *)
	{attribute 'hide'}
	METHOD FB_init : BOOL
	VAR_INPUT
		(*  if TRUE, the retain variables are initialized (warm start / cold start) *)
		bInitRetains : BOOL;
		(*  if TRUE, the instance afterwards gets moved into the copy code (online change) *)
		bInCopyCode : BOOL;
	END_VAR
END_METHOD

END_FUNCTION_BLOCK

// Function Blocks/Camera Register Access/FB_VN_WriteRegister_REAL

	{attribute 'c++_compatible'}
	{attribute 'external_name' := 'FB_VN_WriteRegister_REAL_GUID_172DECAC_D16F_50CA_64B4_5527B069C2B1'}
	{attribute 'TcIecLibraryType'}
	(* This FB writes a REAL value into a register on the camera. Requires an open control channel (e.g. by calling FB_VN_GevCameraControl.OpenCamera() before) *)
	FUNCTION_BLOCK FB_VN_WriteRegister_REAL
	VAR_INPUT
		(* The address of the register that should be written *)
		 {attribute 'GUID' := 'E1ED2436-3512-43FA-B927-3F71DEDDA853'}
		nAddress : GVCP_REGISTER_ADDRESS;
		(* The value to write *)
		fValue : REAL;
		(* OPTIONAL: The endianness of the register. 0 = Big, 1 = Little. Default: 0 *)
		nEndian : UINT;
		(* Writing the register is triggered by a rising edge at this input. *)
		bWrite : BOOL;
	END_VAR
	VAR
		 {attribute 'hide'}
		_reserved1 : USINT;
	END_VAR
	VAR_INPUT
		(* Indicates the time before the function is cancelled. *)
		nTimeout : TIME := VISION_ADS_TIMEOUT;
	END_VAR
	VAR_OUTPUT
		(* This output remains TRUE until the function block has executed a command, but at the longest for the duration supplied to the 'nTimeout' input. While bBusy = TRUE, no new command will be accepted at the inputs. *)
		bBusy : BOOL;
		(* This output is switched to TRUE as soon as an error occurs during the execution of a command. The command-specific error code is contained in ‘nErrorId’. If the function block has a timeout error, 'bError' is TRUE and 'nErrorId' is 1861 (hexadecimal 0x745). Is reset to FALSE by the execution of a command at the inputs. *)
		bError : BOOL;
	END_VAR
	VAR
		 {attribute 'hide'}
		_reserved2 : UINT;
	END_VAR
	VAR_OUTPUT
		(* Contains the ADS error code or the command-specific error code of the last executed command. Is reset to 0 by the execution of a command at the inputs. *)
		nErrorId : UDINT;
	END_VAR
	VAR
		(* Internal reference to the corresponding TcVnGevImageProvider TcCOM module ID, which needs to be set via TC init symbol. *)
		{attribute 'TcInitSymbol'}
		{attribute 'TcCategoryOID' := 'TcVnGevImageProvider'}
		 {attribute 'GUID' := '18071995-0000-0000-0000-00000000000F'}
		oidITcVnGevImageProvider : OTCID;
		 {attribute 'hide'}
		_reserved3 : UINT_0_32;
		(* Internal reference to the corresponding TcVnGevImageProvider module. *)
		{attribute 'hide'}
		 {attribute 'GUID' := 'ED7659DB-95DC-4A4A-B62F-02C9870D5E81'}
		ipGevImageProvider : ITcVnGevImageProvider;
		(* Internal timestamp for timeout detection *)
		{attribute 'hide'}
		nTimeElapsed : TIME;
		(* Internal flag for rising edge detection *)
		{attribute 'hide'}
		bLastWrite : BOOL;
		 {attribute 'hide'}
		_reserved4 : ARRAY [1..3] OF USINT;
	END_VAR


	(* Internal method *)
	{attribute 'hide'}
	METHOD FB_exit : BOOL
	VAR_INPUT
		(*  if TRUE, the exit method is called for exiting an instance that is copied afterwards (online change). *)
		bInCopyCode : BOOL;
	END_VAR
END_METHOD


	(* Internal method *)
	{attribute 'hide'}
	METHOD FB_init : BOOL
	VAR_INPUT
		(*  if TRUE, the retain variables are initialized (warm start / cold start) *)
		bInitRetains : BOOL;
		(*  if TRUE, the instance afterwards gets moved into the copy code (online change) *)
		bInCopyCode : BOOL;
	END_VAR
END_METHOD

END_FUNCTION_BLOCK

// Functions/Control Functions/F_VN_StartAbsWatchdog

	{attribute 'TcIecLibraryType'}
	{attribute 'external_name' := 'F_VN_StartAbsWatchdog_GUID_B6642CE7_60E3_5B20_548C_09E82E542A6F'}
	(* Starts a cooperative watchdog given an absolute stop time. *)
	FUNCTION F_VN_StartAbsWatchdog : HRESULT
	VAR_INPUT
		tStop	:	DINT;	(* Stop time in us *)
		hrPrev	:	HRESULT;	(* HRESULT indicating the result of previous operations (If SUCCEEDED(hrPrev) equals false, no operation is executed.) *)
	END_VAR

END_FUNCTION

// Functions/Control Functions/F_VN_StartAbsWatchdogExp

	{attribute 'TcIecLibraryType'}
	{attribute 'external_name' := 'F_VN_StartAbsWatchdogExp_GUID_262EDCB2_27AA_57B4_7939_97BE3CE24FB9'}
	(* Start a cooperative watchdog given an absolute stop time. (expert function) *)
	FUNCTION F_VN_StartAbsWatchdogExp : HRESULT
	VAR_INPUT
		tStop	:	DINT;	(* Stop time in us *)
		eWatchdogAccType	:	ETcWatchdogAccumulationType;	(* Accumalation method used for combining the results of multiple functions enclosed by this watchdog *)
		hrPrev	:	HRESULT;	(* HRESULT indicating the result of previous operations (If SUCCEEDED(hrPrev) equals false, no operation is executed.) *)
	END_VAR

END_FUNCTION

// Functions/Control Functions/F_VN_StartRelWatchdog

	{attribute 'TcIecLibraryType'}
	{attribute 'external_name' := 'F_VN_StartRelWatchdog_GUID_4DE7377E_52D3_5570_7315_49DAE4E50120'}
	(* Starts a cooperative watchdog given a stop time relative to the current time. *)
	FUNCTION F_VN_StartRelWatchdog : HRESULT
	VAR_INPUT
		tStop	:	DINT;	(* Stop time in us *)
		hrPrev	:	HRESULT;	(* HRESULT indicating the result of previous operations (If SUCCEEDED(hrPrev) equals false, no operation is executed.) *)
	END_VAR

END_FUNCTION

// Functions/Control Functions/F_VN_StartRelWatchdogExp

	{attribute 'TcIecLibraryType'}
	{attribute 'external_name' := 'F_VN_StartRelWatchdogExp_GUID_4EA7FA08_D075_5F40_56BA_CD51E194D939'}
	(* Start a cooperative watchdog given a stop time relative to the current time. (expert function) *)
	FUNCTION F_VN_StartRelWatchdogExp : HRESULT
	VAR_INPUT
		tStop	:	DINT;	(* Stop time in us *)
		eWatchdogAccType	:	ETcWatchdogAccumulationType;	(* Accumalation method used for combining the results of multiple functions enclosed by this watchdog *)
		hrPrev	:	HRESULT;	(* HRESULT indicating the result of previous operations (If SUCCEEDED(hrPrev) equals false, no operation is executed.) *)
	END_VAR

END_FUNCTION

// Functions/Control Functions/F_VN_StopWatchdog

	{attribute 'TcIecLibraryType'}
	{attribute 'external_name' := 'F_VN_StopWatchdog_GUID_243F59AE_3C48_54C1_6F56_DBB4C0B71AAA'}
	(* Stops a watchdog and provide runtime information. *)
	FUNCTION F_VN_StopWatchdog : HRESULT
	VAR_INPUT
		hrStartWatchdog	:	HRESULT;	(* HRESULT indicating the result of the function used to start the watchdog (If SUCCEEDED(hrStartWatchdog) equals false, no operation is executed.) *)
	END_VAR
	VAR_OUTPUT
		nFunctionsMonitored	:	ULINT;	(* Returns the number of functions monitored *)
		nFractionProcessed	:	UDINT;	(* Returns the fraction processed accumulated over the monitored functions in percent *)
		tRest	:	DINT;	(* Returns the remaining computation time in us (may be negative) *)
	END_VAR

END_FUNCTION

// Functions/Image Segmentation/F_VN_AdaptiveThreshold

	{attribute 'TcIecLibraryType'}
	{attribute 'external_name' := 'F_VN_AdaptiveThreshold_GUID_CA6B0105_B730_5DEC_6046_F20276E17033'}
	(* Apply an adaptive threshold to a gray level image. *)
	FUNCTION F_VN_AdaptiveThreshold : HRESULT
	VAR_INPUT
		ipSrcImage	:	ITcVnImage;	(* Source image (1 channel, elements of type USINT) *)
		ipDestImage	:	REFERENCE TO ITcVnImage;	(* Destination image (An appropriate destination image will be created if required.) *)
		fMaxValue	:	LREAL;	(* Value assigned to pixels for which the threshold condition is true *)
		hrPrev	:	HRESULT;	(* HRESULT indicating the result of previous operations (If SUCCEEDED(hrPrev) equals false, no operation is executed.) *)
	END_VAR

END_FUNCTION

// Functions/Image Segmentation/F_VN_AdaptiveThresholdExp

	{attribute 'TcIecLibraryType'}
	{attribute 'external_name' := 'F_VN_AdaptiveThresholdExp_GUID_9FC98429_48DD_59EA_6774_51D8412A4317'}
	(* Apply an adaptive threshold to a gray level image. (expert function) *)
	FUNCTION F_VN_AdaptiveThresholdExp : HRESULT
	VAR_INPUT
		ipSrcImage	:	ITcVnImage;	(* Source image (1 channel, elements of type USINT) *)
		ipDestImage	:	REFERENCE TO ITcVnImage;	(* Destination image (An appropriate destination image will be created if required.) *)
		fMaxValue	:	LREAL;	(* Value assigned to pixels for which the threshold condition is true *)
		eAdaptiveMethod	:	ETcVnAdaptiveThresholdMethod;	(* Adaptive threshold method to be applied (MEAN: threshold value will be calculated as a mean of the nBlockSize x nBlockSize neighborhood of (x,y) minus fConstant. GAUSSIAN: threshold value is a weighted sum (cross-correlation with a Gaussian window) of the nBlockSize x nBlockSize neighborhood of (x,y) minus fConstant. *)
		eThresholdType	:	ETcVnThresholdType;	(* Threshold type to be applied (only BINARY and BINARY_INV are supported) *)
		nBlockSize	:	UDINT;	(* Size of the pixel neighborhood to calculate the local threshold (3, 5, 7, ...) *)
		fConstant	:	LREAL;	(* Constant that is subtracted from the weighted mean of the pixel neighborhood, which leads to the local threshold *)
		hrPrev	:	HRESULT;	(* HRESULT indicating the result of previous operations (If SUCCEEDED(hrPrev) equals false, no operation is executed.) *)
	END_VAR

END_FUNCTION

// Functions/Image Segmentation/F_VN_CheckColorRange

	{attribute 'TcIecLibraryType'}
	{attribute 'external_name' := 'F_VN_CheckColorRange_GUID_24D2EC60_0C87_5741_7363_F4F8B428217B'}
	(* Check if the pixel values of an image lie in a given range. The destination image has the same size as the source image but only one channel with
          a pixel element size of 8 bit. Its elements are set to 255 if the corresponding pixels of the source image are in the checked range and set to 0 otherwise. *)
	FUNCTION F_VN_CheckColorRange : HRESULT
	VAR_INPUT
		ipSrcImage	:	ITcVnImage;	(* Source image *)
		ipDestImage	:	REFERENCE TO ITcVnImage;	(* Destination image (An appropriate destination image will be created if required.) *)
		aLowerBounds	:	REFERENCE TO TcVnVector4_LREAL;	(* Channel-wise lower bounds (Unused channels are ignored.) *)
		aUpperBounds	:	REFERENCE TO TcVnVector4_LREAL;	(* Channel-wise upper bounds (Unused channels are ignored.) *)
		hrPrev	:	HRESULT;	(* HRESULT indicating the result of previous operations (If SUCCEEDED(hrPrev) equals false, no operation is executed.) *)
	END_VAR

END_FUNCTION

// Functions/Image Segmentation/F_VN_Threshold

	{attribute 'TcIecLibraryType'}
	{attribute 'external_name' := 'F_VN_Threshold_GUID_8F68F06A_5695_564C_5744_5F520510FFD6'}
	(* Apply a fixed threshold or a dynamic threshold according to Otsu. *)
	FUNCTION F_VN_Threshold : HRESULT
	VAR_INPUT
		ipSrcImage	:	ITcVnImage;	(* Source image (For Otsu and Triangle threshold types, only 1 channel of TCVN_ET_USINT is supported) *)
		ipDestImage	:	REFERENCE TO ITcVnImage;	(* Destination image (An appropriate destination image will be created if required.) *)
		fThreshold	:	LREAL;	(* Fixed threshold (unused if dynamic thresholding is selected) *)
		fMaxValue	:	LREAL;	(* Maximum pixel value *)
		eThresholdType	:	ETcVnThresholdType;	(* Threshold type to be applied *)
		hrPrev	:	HRESULT;	(* HRESULT indicating the result of previous operations (If SUCCEEDED(hrPrev) equals false, no operation is executed.) *)
	END_VAR

END_FUNCTION

// Functions/Image Segmentation/F_VN_WatershedSegmentationExp

	{attribute 'TcIecLibraryType'}
	{attribute 'external_name' := 'F_VN_WatershedSegmentationExp_GUID_7E933569_D82C_5D67_59F2_B27A74CFF7E5'}
	(* Apply a marker-based watershed segmentation. (expert function) *)
	FUNCTION F_VN_WatershedSegmentationExp : HRESULT
	VAR_INPUT
		ipSrcImage	:	ITcVnImage;	(* Source image (USINT, 3 channels) *)
		ipDestImage	:	REFERENCE TO ITcVnImage;	(* Destination image (DINT, 1 channel. An appropriate image will be created if required.) *)
		ipMarkers	:	ITcVnImage;	(* Marker image (DINT, 1 channel) *)
		hrPrev	:	HRESULT;	(* HRESULT indicating the result of previous operations (If SUCCEEDED(hrPrev) equals false, no operation is executed.) *)
	END_VAR

END_FUNCTION

// Functions/Algebraic Container Operations/F_VN_AddContainers

	{attribute 'TcIecLibraryType'}
	{attribute 'external_name' := 'F_VN_AddContainers_GUID_4F1F15AF_95B5_56E0_6213_64A95096DD5F'}
	(* Element-wise addition of two containers (same length and type). *)
	FUNCTION F_VN_AddContainers : HRESULT
	VAR_INPUT
		ipSrcContainer1	:	ITcVnContainer;	(* Source container 1 *)
		ipSrcContainer2	:	ITcVnContainer;	(* Source container 2 *)
		ipDestContainer	:	REFERENCE TO ITcVnContainer;	(* Returns the resulting container *)
		hrPrev	:	HRESULT;	(* HRESULT indicating the result of previous operations (If SUCCEEDED(hrPrev) equals false, no operation is executed.) *)
	END_VAR

END_FUNCTION

// Functions/Algebraic Container Operations/F_VN_BitwiseAndContainers

	{attribute 'TcIecLibraryType'}
	{attribute 'external_name' := 'F_VN_BitwiseAndContainers_GUID_90A20C65_B315_563E_73B6_B2080C88FC63'}
	(* Element-wise application of a bit-wise AND operator to two containers (same length and type, integer only). *)
	FUNCTION F_VN_BitwiseAndContainers : HRESULT
	VAR_INPUT
		ipSrcContainer1	:	ITcVnContainer;	(* Source container 1 *)
		ipSrcContainer2	:	ITcVnContainer;	(* Source container 2 *)
		ipDestContainer	:	REFERENCE TO ITcVnContainer;	(* Returns the resulting container *)
		hrPrev	:	HRESULT;	(* HRESULT indicating the result of previous operations (If SUCCEEDED(hrPrev) equals false, no operation is executed.) *)
	END_VAR

END_FUNCTION

// Functions/Algebraic Container Operations/F_VN_BitwiseNotContainer

	{attribute 'TcIecLibraryType'}
	{attribute 'external_name' := 'F_VN_BitwiseNotContainer_GUID_8CC31781_7A10_5E0D_7461_661E89417142'}
	(* Element-wise application of a bit-wise NOT operator to a container (integer only). *)
	FUNCTION F_VN_BitwiseNotContainer : HRESULT
	VAR_INPUT
		ipSrcContainer	:	ITcVnContainer;	(* Source container *)
		ipDestContainer	:	REFERENCE TO ITcVnContainer;	(* Returns the resulting container *)
		hrPrev	:	HRESULT;	(* HRESULT indicating the result of previous operations (If SUCCEEDED(hrPrev) equals false, no operation is executed.) *)
	END_VAR

END_FUNCTION

// Functions/Algebraic Container Operations/F_VN_BitwiseOrContainers

	{attribute 'TcIecLibraryType'}
	{attribute 'external_name' := 'F_VN_BitwiseOrContainers_GUID_8BA48D59_D1BC_5E8A_640B_52D609BD74B1'}
	(* Element-wise application of a bit-wise OR operator to two containers (same length and type, integer only). *)
	FUNCTION F_VN_BitwiseOrContainers : HRESULT
	VAR_INPUT
		ipSrcContainer1	:	ITcVnContainer;	(* Source container 1 *)
		ipSrcContainer2	:	ITcVnContainer;	(* Source container 2 *)
		ipDestContainer	:	REFERENCE TO ITcVnContainer;	(* Returns the resulting container *)
		hrPrev	:	HRESULT;	(* HRESULT indicating the result of previous operations (If SUCCEEDED(hrPrev) equals false, no operation is executed.) *)
	END_VAR

END_FUNCTION

// Functions/Algebraic Container Operations/F_VN_BitwiseXorContainers

	{attribute 'TcIecLibraryType'}
	{attribute 'external_name' := 'F_VN_BitwiseXorContainers_GUID_CBDD7338_BF69_5B44_7EB6_739B94CEB669'}
	(* Element-wise application of a bit-wise XOR operator to two containers (same length and type, integer only). *)
	FUNCTION F_VN_BitwiseXorContainers : HRESULT
	VAR_INPUT
		ipSrcContainer1	:	ITcVnContainer;	(* Source container 1 *)
		ipSrcContainer2	:	ITcVnContainer;	(* Source container 2 *)
		ipDestContainer	:	REFERENCE TO ITcVnContainer;	(* Returns the resulting container *)
		hrPrev	:	HRESULT;	(* HRESULT indicating the result of previous operations (If SUCCEEDED(hrPrev) equals false, no operation is executed.) *)
	END_VAR

END_FUNCTION

// Functions/Algebraic Container Operations/F_VN_DivideContainers

	{attribute 'TcIecLibraryType'}
	{attribute 'external_name' := 'F_VN_DivideContainers_GUID_34AD89ED_1379_542C_690B_4959A815EF32'}
	(* Element-wise division of two containers (same length and type). In case of integer division by zero, the resulting element is set to 0 and S_DIVISION_BY_ZERO is returned instead of S_OK (value can be changed in F_VN_DivideContainersExp). *)
	FUNCTION F_VN_DivideContainers : HRESULT
	VAR_INPUT
		ipSrcContainer1	:	ITcVnContainer;	(* Source container 1 *)
		ipSrcContainer2	:	ITcVnContainer;	(* Source container 2 *)
		ipDestContainer	:	REFERENCE TO ITcVnContainer;	(* Returns the resulting container *)
		hrPrev	:	HRESULT;	(* HRESULT indicating the result of previous operations (If SUCCEEDED(hrPrev) equals false, no operation is executed.) *)
	END_VAR

END_FUNCTION

// Functions/Algebraic Container Operations/F_VN_DivideContainersExp

	{attribute 'TcIecLibraryType'}
	{attribute 'external_name' := 'F_VN_DivideContainersExp_GUID_2CB04FFF_D1DA_5A0E_516E_F5768FDB5A7F'}
	(* Element-wise division of two containers (same length and type). In case of integer division by zero, the resulting element is set to nIntDivideByZeroResult and S_DIVISION_BY_ZERO is returned instead of S_OK. (expert function) *)
	FUNCTION F_VN_DivideContainersExp : HRESULT
	VAR_INPUT
		ipSrcContainer1	:	ITcVnContainer;	(* Source container 1 *)
		ipSrcContainer2	:	ITcVnContainer;	(* Source container 2 *)
		ipDestContainer	:	REFERENCE TO ITcVnContainer;	(* Returns the resulting container *)
		nIntDivideByZeroResult	:	LINT;	(* Value set as result in case of integer division by zero *)
		hrPrev	:	HRESULT;	(* HRESULT indicating the result of previous operations (If SUCCEEDED(hrPrev) equals false, no operation is executed.) *)
	END_VAR

END_FUNCTION

// Functions/Algebraic Container Operations/F_VN_MaxContainer

	{attribute 'TcIecLibraryType'}
	{attribute 'external_name' := 'F_VN_MaxContainer_GUID_FC30E752_0F2A_5867_6812_9FE61E61F698'}
	(* Element-wise maximum of two containers (same length and type). *)
	FUNCTION F_VN_MaxContainer : HRESULT
	VAR_INPUT
		ipSrcContainer1	:	ITcVnContainer;	(* Source container 1 *)
		ipSrcContainer2	:	ITcVnContainer;	(* Source container 2 *)
		ipDestContainer	:	REFERENCE TO ITcVnContainer;	(* Returns the resulting container *)
		hrPrev	:	HRESULT;	(* HRESULT indicating the result of previous operations (If SUCCEEDED(hrPrev) equals false, no operation is executed.) *)
	END_VAR

END_FUNCTION

// Functions/Algebraic Container Operations/F_VN_MinContainer

	{attribute 'TcIecLibraryType'}
	{attribute 'external_name' := 'F_VN_MinContainer_GUID_76517ED0_EA82_5E07_53D0_B4F7C4F578AC'}
	(* Element-wise minimum of two containers (same length and type). *)
	FUNCTION F_VN_MinContainer : HRESULT
	VAR_INPUT
		ipSrcContainer1	:	ITcVnContainer;	(* Source container 1 *)
		ipSrcContainer2	:	ITcVnContainer;	(* Source container 2 *)
		ipDestContainer	:	REFERENCE TO ITcVnContainer;	(* Returns the resulting container *)
		hrPrev	:	HRESULT;	(* HRESULT indicating the result of previous operations (If SUCCEEDED(hrPrev) equals false, no operation is executed.) *)
	END_VAR

END_FUNCTION

// Functions/Algebraic Container Operations/F_VN_MultiplyContainers

	{attribute 'TcIecLibraryType'}
	{attribute 'external_name' := 'F_VN_MultiplyContainers_GUID_6EEB615B_6FA7_5AC3_6948_BD220FEFCD09'}
	(* Element-wise multiplication of two containers (same length and type). *)
	FUNCTION F_VN_MultiplyContainers : HRESULT
	VAR_INPUT
		ipSrcContainer1	:	ITcVnContainer;	(* Source container 1 *)
		ipSrcContainer2	:	ITcVnContainer;	(* Source container 2 *)
		ipDestContainer	:	REFERENCE TO ITcVnContainer;	(* Returns the resulting container *)
		hrPrev	:	HRESULT;	(* HRESULT indicating the result of previous operations (If SUCCEEDED(hrPrev) equals false, no operation is executed.) *)
	END_VAR

END_FUNCTION

// Functions/Algebraic Container Operations/F_VN_NegateContainer

	{attribute 'TcIecLibraryType'}
	{attribute 'external_name' := 'F_VN_NegateContainer_GUID_7C324A98_063B_51BB_78E2_3FAE943CB90F'}
	(* Element-wise negation of a container (two's complement). *)
	FUNCTION F_VN_NegateContainer : HRESULT
	VAR_INPUT
		ipSrcContainer	:	ITcVnContainer;	(* Source container *)
		ipDestContainer	:	REFERENCE TO ITcVnContainer;	(* Returns the resulting container (same type as ipSrcContainer) *)
		hrPrev	:	HRESULT;	(* HRESULT indicating the result of previous operations (If SUCCEEDED(hrPrev) equals false, no operation is executed.) *)
	END_VAR

END_FUNCTION

// Functions/Algebraic Container Operations/F_VN_SubtractContainers

	{attribute 'TcIecLibraryType'}
	{attribute 'external_name' := 'F_VN_SubtractContainers_GUID_567E8307_F10D_58D4_6587_7E1D833A1546'}
	(* Element-wise subtraction of two containers (same length and type). *)
	FUNCTION F_VN_SubtractContainers : HRESULT
	VAR_INPUT
		ipSrcContainer1	:	ITcVnContainer;	(* Source container 1 *)
		ipSrcContainer2	:	ITcVnContainer;	(* Source container 2 *)
		ipDestContainer	:	REFERENCE TO ITcVnContainer;	(* Returns the resulting container *)
		hrPrev	:	HRESULT;	(* HRESULT indicating the result of previous operations (If SUCCEEDED(hrPrev) equals false, no operation is executed.) *)
	END_VAR

END_FUNCTION

// Functions/Algebraic Image Operations/F_VN_AddImages

	{attribute 'TcIecLibraryType'}
	{attribute 'external_name' := 'F_VN_AddImages_GUID_1F1D8C7E_08BE_5BBF_47B6_CA42AD7489EB'}
	(* Element-wise addition of two images using saturation arithmetics. *)
	FUNCTION F_VN_AddImages : HRESULT
	VAR_INPUT
		ipSrcImage1	:	ITcVnImage;	(* First source image *)
		ipSrcImage2	:	ITcVnImage;	(* Second source image *)
		ipDestImage	:	REFERENCE TO ITcVnImage;	(* Destination image (An appropriate destination image will be created if required.) *)
		hrPrev	:	HRESULT;	(* HRESULT indicating the result of previous operations (If SUCCEEDED(hrPrev) equals false, no operation is executed.) *)
	END_VAR

END_FUNCTION

// Functions/Algebraic Image Operations/F_VN_AddScalarToImage

	{attribute 'TcIecLibraryType'}
	{attribute 'external_name' := 'F_VN_AddScalarToImage_GUID_33D8530F_424C_5B78_530B_DD1D571B70C7'}
	(* Add a scalar value to each image pixel using saturation arithmetics. *)
	FUNCTION F_VN_AddScalarToImage : HRESULT
	VAR_INPUT
		fScalar	:	LREAL;	(* Scalar value *)
		ipSrcImage	:	ITcVnImage;	(* Source image *)
		ipDestImage	:	REFERENCE TO ITcVnImage;	(* Destination image (An appropriate destination image will be created if required.) *)
		hrPrev	:	HRESULT;	(* HRESULT indicating the result of previous operations (If SUCCEEDED(hrPrev) equals false, no operation is executed.) *)
	END_VAR

END_FUNCTION

// Functions/Algebraic Image Operations/F_VN_AddVectorToImage

	{attribute 'TcIecLibraryType'}
	{attribute 'external_name' := 'F_VN_AddVectorToImage_GUID_A6AF7B1B_8B45_5EBA_50CA_20B242C7DB45'}
	(* Add a vector (1 element for each image channel) to each image pixel using saturation arithmetics. *)
	FUNCTION F_VN_AddVectorToImage : HRESULT
	VAR_INPUT
		aVector	:	REFERENCE TO TcVnVector4_LREAL;	(* 4-element vector (1 element for each image channel. If the image has less channels, the further vector elements are ignored.) *)
		ipSrcImage	:	ITcVnImage;	(* Source image *)
		ipDestImage	:	REFERENCE TO ITcVnImage;	(* Destination image (An appropriate destination image will be created if required.) *)
		hrPrev	:	HRESULT;	(* HRESULT indicating the result of previous operations (If SUCCEEDED(hrPrev) equals false, no operation is executed.) *)
	END_VAR

END_FUNCTION

// Functions/Algebraic Image Operations/F_VN_BitwiseAndImages

	{attribute 'TcIecLibraryType'}
	{attribute 'external_name' := 'F_VN_BitwiseAndImages_GUID_C504C846_5E8A_5008_4C2C_85F74D342004'}
	(* Element-wise application of a bit-wise AND operator to two images. *)
	FUNCTION F_VN_BitwiseAndImages : HRESULT
	VAR_INPUT
		ipSrcImage1	:	ITcVnImage;	(* First source image *)
		ipSrcImage2	:	ITcVnImage;	(* Second source image *)
		ipDestImage	:	REFERENCE TO ITcVnImage;	(* Destination image (An appropriate destination image will be created if required.) *)
		hrPrev	:	HRESULT;	(* HRESULT indicating the result of previous operations (If SUCCEEDED(hrPrev) equals false, no operation is executed.) *)
	END_VAR

END_FUNCTION

// Functions/Algebraic Image Operations/F_VN_BitwiseAndImagesExp

	{attribute 'TcIecLibraryType'}
	{attribute 'external_name' := 'F_VN_BitwiseAndImagesExp_GUID_53FE7276_649E_5300_79E0_80223D84D7E3'}
	(* Element-wise application of a bit-wise AND operator to two images. (expert function) *)
	FUNCTION F_VN_BitwiseAndImagesExp : HRESULT
	VAR_INPUT
		ipSrcImage1	:	ITcVnImage;	(* First source image *)
		ipSrcImage2	:	ITcVnImage;	(* Second source image *)
		ipDestImage	:	REFERENCE TO ITcVnImage;	(* Destination image (An appropriate destination image will be created if required.) *)
		ipMask	:	ITcVnImage;	(* Mask to limit the operation to specific pixel positions (mask value 0: skip pixel, mask value > 0: apply operation to pixel) *)
		hrPrev	:	HRESULT;	(* HRESULT indicating the result of previous operations (If SUCCEEDED(hrPrev) equals false, no operation is executed.) *)
	END_VAR

END_FUNCTION

// Functions/Algebraic Image Operations/F_VN_BitwiseAndScalarWithImage

	{attribute 'TcIecLibraryType'}
	{attribute 'external_name' := 'F_VN_BitwiseAndScalarWithImage_GUID_4388DF1A_75E7_5F46_5F83_80F8DE8A19AC'}
	(* Bitwise and a scalar value with each image pixel. *)
	FUNCTION F_VN_BitwiseAndScalarWithImage : HRESULT
	VAR_INPUT
		fScalar	:	LREAL;	(* Scalar value *)
		ipSrcImage	:	ITcVnImage;	(* Source image *)
		ipDestImage	:	REFERENCE TO ITcVnImage;	(* Destination image (An appropriate destination image will be created if required.) *)
		hrPrev	:	HRESULT;	(* HRESULT indicating the result of previous operations (If SUCCEEDED(hrPrev) equals false, no operation is executed.) *)
	END_VAR

END_FUNCTION

// Functions/Algebraic Image Operations/F_VN_BitwiseAndVectorWithImage

	{attribute 'TcIecLibraryType'}
	{attribute 'external_name' := 'F_VN_BitwiseAndVectorWithImage_GUID_4744945F_C8DD_566D_6067_C2E170DE3155'}
	(* Bitwise and a vector (1 element for each image channel) with each image pixel. *)
	FUNCTION F_VN_BitwiseAndVectorWithImage : HRESULT
	VAR_INPUT
		aVector	:	REFERENCE TO TcVnVector4_LREAL;	(* 4-element vector (1 element for each image channel. If the image has less channels, the further vector elements are ignored.) *)
		ipSrcImage	:	ITcVnImage;	(* Source image *)
		ipDestImage	:	REFERENCE TO ITcVnImage;	(* Destination image (An appropriate destination image will be created if required.) *)
		hrPrev	:	HRESULT;	(* HRESULT indicating the result of previous operations (If SUCCEEDED(hrPrev) equals false, no operation is executed.) *)
	END_VAR

END_FUNCTION

// Functions/Algebraic Image Operations/F_VN_BitwiseNotImage

	{attribute 'TcIecLibraryType'}
	{attribute 'external_name' := 'F_VN_BitwiseNotImage_GUID_7FB2FED1_F387_5D78_49A9_441E0902CFB1'}
	(* Element-wise application of a bit-wise NOT operator to an image. *)
	FUNCTION F_VN_BitwiseNotImage : HRESULT
	VAR_INPUT
		ipSrcImage	:	ITcVnImage;	(* Source image *)
		ipDestImage	:	REFERENCE TO ITcVnImage;	(* Destination image (An appropriate destination image will be created if required.) *)
		hrPrev	:	HRESULT;	(* HRESULT indicating the result of previous operations (If SUCCEEDED(hrPrev) equals false, no operation is executed.) *)
	END_VAR

END_FUNCTION

// Functions/Algebraic Image Operations/F_VN_BitwiseNotImageExp

	{attribute 'TcIecLibraryType'}
	{attribute 'external_name' := 'F_VN_BitwiseNotImageExp_GUID_41CD1509_8DBB_52EA_7C26_DF3D56CF6622'}
	(* Element-wise application of a bit-wise NOT operator to an image. (expert function) *)
	FUNCTION F_VN_BitwiseNotImageExp : HRESULT
	VAR_INPUT
		ipSrcImage	:	ITcVnImage;	(* Source image *)
		ipDestImage	:	REFERENCE TO ITcVnImage;	(* Destination image (An appropriate destination image will be created if required.) *)
		ipMask	:	ITcVnImage;	(* Mask to limit the operation to specific pixel positions (mask value 0: skip pixel, mask value > 0: apply operation to pixel) *)
		hrPrev	:	HRESULT;	(* HRESULT indicating the result of previous operations (If SUCCEEDED(hrPrev) equals false, no operation is executed.) *)
	END_VAR

END_FUNCTION

// Functions/Algebraic Image Operations/F_VN_BitwiseOrImages

	{attribute 'TcIecLibraryType'}
	{attribute 'external_name' := 'F_VN_BitwiseOrImages_GUID_B21FC762_1392_5F1C_6D12_3AF7DA91C375'}
	(* Element-wise application of a bit-wise OR operator to two images. *)
	FUNCTION F_VN_BitwiseOrImages : HRESULT
	VAR_INPUT
		ipSrcImage1	:	ITcVnImage;	(* First source image *)
		ipSrcImage2	:	ITcVnImage;	(* Second source image *)
		ipDestImage	:	REFERENCE TO ITcVnImage;	(* Destination image (An appropriate destination image will be created if required.) *)
		hrPrev	:	HRESULT;	(* HRESULT indicating the result of previous operations (If SUCCEEDED(hrPrev) equals false, no operation is executed.) *)
	END_VAR

END_FUNCTION

// Functions/Algebraic Image Operations/F_VN_BitwiseOrImagesExp

	{attribute 'TcIecLibraryType'}
	{attribute 'external_name' := 'F_VN_BitwiseOrImagesExp_GUID_1E51298D_9561_53A5_6634_CD58E7299378'}
	(* Element-wise application of a bit-wise OR operator to two images. (expert function) *)
	FUNCTION F_VN_BitwiseOrImagesExp : HRESULT
	VAR_INPUT
		ipSrcImage1	:	ITcVnImage;	(* First source image *)
		ipSrcImage2	:	ITcVnImage;	(* Second source image *)
		ipDestImage	:	REFERENCE TO ITcVnImage;	(* Destination image (An appropriate destination image will be created if required.) *)
		ipMask	:	ITcVnImage;	(* Mask to limit the operation to specific pixel positions (mask value 0: skip pixel, mask value > 0: apply operation to pixel) *)
		hrPrev	:	HRESULT;	(* HRESULT indicating the result of previous operations (If SUCCEEDED(hrPrev) equals false, no operation is executed.) *)
	END_VAR

END_FUNCTION

// Functions/Algebraic Image Operations/F_VN_BitwiseOrScalarWithImage

	{attribute 'TcIecLibraryType'}
	{attribute 'external_name' := 'F_VN_BitwiseOrScalarWithImage_GUID_749A4B55_9C76_5C0B_7A08_8EF6FD3214FF'}
	(* Bitwise or a scalar value with each image pixel. *)
	FUNCTION F_VN_BitwiseOrScalarWithImage : HRESULT
	VAR_INPUT
		fScalar	:	LREAL;	(* Scalar value *)
		ipSrcImage	:	ITcVnImage;	(* Source image *)
		ipDestImage	:	REFERENCE TO ITcVnImage;	(* Destination image (An appropriate destination image will be created if required.) *)
		hrPrev	:	HRESULT;	(* HRESULT indicating the result of previous operations (If SUCCEEDED(hrPrev) equals false, no operation is executed.) *)
	END_VAR

END_FUNCTION

// Functions/Algebraic Image Operations/F_VN_BitwiseOrVectorWithImage

	{attribute 'TcIecLibraryType'}
	{attribute 'external_name' := 'F_VN_BitwiseOrVectorWithImage_GUID_3342CE5C_46EC_5157_58F6_126F0D1C915A'}
	(* Bitwise or a vector (1 element for each image channel) with each image pixel. *)
	FUNCTION F_VN_BitwiseOrVectorWithImage : HRESULT
	VAR_INPUT
		aVector	:	REFERENCE TO TcVnVector4_LREAL;	(* 4-element vector (1 element for each image channel. If the image has less channels, the further vector elements are ignored.) *)
		ipSrcImage	:	ITcVnImage;	(* Source image *)
		ipDestImage	:	REFERENCE TO ITcVnImage;	(* Destination image (An appropriate destination image will be created if required.) *)
		hrPrev	:	HRESULT;	(* HRESULT indicating the result of previous operations (If SUCCEEDED(hrPrev) equals false, no operation is executed.) *)
	END_VAR

END_FUNCTION

// Functions/Algebraic Image Operations/F_VN_BitwiseXorImages

	{attribute 'TcIecLibraryType'}
	{attribute 'external_name' := 'F_VN_BitwiseXorImages_GUID_73A7C128_E190_5F68_6711_1E8D04C2E8A0'}
	(* Element-wise application of a bit-wise XOR operator to two images. *)
	FUNCTION F_VN_BitwiseXorImages : HRESULT
	VAR_INPUT
		ipSrcImage1	:	ITcVnImage;	(* First source image *)
		ipSrcImage2	:	ITcVnImage;	(* Second source image *)
		ipDestImage	:	REFERENCE TO ITcVnImage;	(* Destination image (An appropriate destination image will be created if required.) *)
		hrPrev	:	HRESULT;	(* HRESULT indicating the result of previous operations (If SUCCEEDED(hrPrev) equals false, no operation is executed.) *)
	END_VAR

END_FUNCTION

// Functions/Algebraic Image Operations/F_VN_BitwiseXorImagesExp

	{attribute 'TcIecLibraryType'}
	{attribute 'external_name' := 'F_VN_BitwiseXorImagesExp_GUID_20E66FD2_A099_597C_52F2_74B86A085671'}
	(* Element-wise application of a bit-wise XOR operator to two images. (expert function) *)
	FUNCTION F_VN_BitwiseXorImagesExp : HRESULT
	VAR_INPUT
		ipSrcImage1	:	ITcVnImage;	(* First source image *)
		ipSrcImage2	:	ITcVnImage;	(* Second source image *)
		ipDestImage	:	REFERENCE TO ITcVnImage;	(* Destination image (An appropriate destination image will be created if required.) *)
		ipMask	:	ITcVnImage;	(* Mask to limit the operation to specific pixel positions (mask value 0: skip pixel, mask value > 0: apply operation to pixel) *)
		hrPrev	:	HRESULT;	(* HRESULT indicating the result of previous operations (If SUCCEEDED(hrPrev) equals false, no operation is executed.) *)
	END_VAR

END_FUNCTION

// Functions/Algebraic Image Operations/F_VN_BitwiseXorScalarWithImage

	{attribute 'TcIecLibraryType'}
	{attribute 'external_name' := 'F_VN_BitwiseXorScalarWithImage_GUID_4A6386BC_7A04_581B_40F8_BFCA2B05001E'}
	(* Bitwise xor a scalar value with each image pixel. *)
	FUNCTION F_VN_BitwiseXorScalarWithImage : HRESULT
	VAR_INPUT
		fScalar	:	LREAL;	(* Scalar value *)
		ipSrcImage	:	ITcVnImage;	(* Source image *)
		ipDestImage	:	REFERENCE TO ITcVnImage;	(* Destination image (An appropriate destination image will be created if required.) *)
		hrPrev	:	HRESULT;	(* HRESULT indicating the result of previous operations (If SUCCEEDED(hrPrev) equals false, no operation is executed.) *)
	END_VAR

END_FUNCTION

// Functions/Algebraic Image Operations/F_VN_BitwiseXorVectorWithImage

	{attribute 'TcIecLibraryType'}
	{attribute 'external_name' := 'F_VN_BitwiseXorVectorWithImage_GUID_CC153B56_F703_5887_44B2_B9059F07BC39'}
	(* Bitwise xor a vector (1 element for each image channel) with each image pixel. *)
	FUNCTION F_VN_BitwiseXorVectorWithImage : HRESULT
	VAR_INPUT
		aVector	:	REFERENCE TO TcVnVector4_LREAL;	(* 4-element vector (1 element for each image channel. If the image has less channels, the further vector elements are ignored.) *)
		ipSrcImage	:	ITcVnImage;	(* Source image *)
		ipDestImage	:	REFERENCE TO ITcVnImage;	(* Destination image (An appropriate destination image will be created if required.) *)
		hrPrev	:	HRESULT;	(* HRESULT indicating the result of previous operations (If SUCCEEDED(hrPrev) equals false, no operation is executed.) *)
	END_VAR

END_FUNCTION

// Functions/Algebraic Image Operations/F_VN_DivideImageByScalar

	{attribute 'TcIecLibraryType'}
	{attribute 'external_name' := 'F_VN_DivideImageByScalar_GUID_63AF1058_8576_57FD_73F1_80A8AF8828F7'}
	(* Divide each image pixel by a scalar value using saturation arithmetics. *)
	FUNCTION F_VN_DivideImageByScalar : HRESULT
	VAR_INPUT
		ipSrcImage	:	ITcVnImage;	(* Source image *)
		fScalar	:	LREAL;	(* Scalar value *)
		ipDestImage	:	REFERENCE TO ITcVnImage;	(* Destination image (An appropriate destination image will be created if required.) *)
		hrPrev	:	HRESULT;	(* HRESULT indicating the result of previous operations (If SUCCEEDED(hrPrev) equals false, no operation is executed.) *)
	END_VAR

END_FUNCTION

// Functions/Algebraic Image Operations/F_VN_DivideImageByVector

	{attribute 'TcIecLibraryType'}
	{attribute 'external_name' := 'F_VN_DivideImageByVector_GUID_9350EECB_F5F0_5A4B_712C_4363426B17BF'}
	(* Divides each image pixel by a vector (1 element for each image channel) using saturation arithmetics. *)
	FUNCTION F_VN_DivideImageByVector : HRESULT
	VAR_INPUT
		ipSrcImage	:	ITcVnImage;	(* Source image *)
		aVector	:	REFERENCE TO TcVnVector4_LREAL;	(* 4-element vector (1 element for each image channel. If the image has less channels, the further vector elements are ignored.) *)
		ipDestImage	:	REFERENCE TO ITcVnImage;	(* Destination image (An appropriate destination image will be created if required.) *)
		hrPrev	:	HRESULT;	(* HRESULT indicating the result of previous operations (If SUCCEEDED(hrPrev) equals false, no operation is executed.) *)
	END_VAR

END_FUNCTION

// Functions/Algebraic Image Operations/F_VN_DivideImages

	{attribute 'TcIecLibraryType'}
	{attribute 'external_name' := 'F_VN_DivideImages_GUID_73A44C60_7FB3_5EC8_7CF3_39CB9018D281'}
	(* Element-wise division of two images using saturation arithmetics. (A division by zero equals zero.) *)
	FUNCTION F_VN_DivideImages : HRESULT
	VAR_INPUT
		ipSrcImage1	:	ITcVnImage;	(* First source image (dividend) *)
		ipSrcImage2	:	ITcVnImage;	(* Second source image (divisor) *)
		ipDestImage	:	REFERENCE TO ITcVnImage;	(* Destination image (An appropriate destination image will be created if required.) *)
		hrPrev	:	HRESULT;	(* HRESULT indicating the result of previous operations (If SUCCEEDED(hrPrev) equals false, no operation is executed.) *)
	END_VAR

END_FUNCTION

// Functions/Algebraic Image Operations/F_VN_DivideScalarByImage

	{attribute 'TcIecLibraryType'}
	{attribute 'external_name' := 'F_VN_DivideScalarByImage_GUID_20D1705D_B1A0_5218_415B_4AECA4CAC8D6'}
	(* Divides a scalar value by each image pixel using saturation arithmetics. *)
	FUNCTION F_VN_DivideScalarByImage : HRESULT
	VAR_INPUT
		fScalar	:	LREAL;	(* Scalar value *)
		ipSrcImage	:	ITcVnImage;	(* Source image *)
		ipDestImage	:	REFERENCE TO ITcVnImage;	(* Destination image (An appropriate destination image will be created if required.) *)
		hrPrev	:	HRESULT;	(* HRESULT indicating the result of previous operations (If SUCCEEDED(hrPrev) equals false, no operation is executed.) *)
	END_VAR

END_FUNCTION

// Functions/Algebraic Image Operations/F_VN_DivideVectorByImage

	{attribute 'TcIecLibraryType'}
	{attribute 'external_name' := 'F_VN_DivideVectorByImage_GUID_2BF41330_876E_561E_7116_0CFD1BFA154E'}
	(* Divides a vector (1 element for each image channel) by each image pixel using saturation arithmetics. *)
	FUNCTION F_VN_DivideVectorByImage : HRESULT
	VAR_INPUT
		aVector	:	REFERENCE TO TcVnVector4_LREAL;	(* 4-element vector (1 element for each image channel. If the image has less channels, the further vector elements are ignored.) *)
		ipSrcImage	:	ITcVnImage;	(* Source image *)
		ipDestImage	:	REFERENCE TO ITcVnImage;	(* Destination image (An appropriate destination image will be created if required.) *)
		hrPrev	:	HRESULT;	(* HRESULT indicating the result of previous operations (If SUCCEEDED(hrPrev) equals false, no operation is executed.) *)
	END_VAR

END_FUNCTION

// Functions/Algebraic Image Operations/F_VN_ElementwiseExp

	{attribute 'TcIecLibraryType'}
	{attribute 'external_name' := 'F_VN_ElementwiseExp_GUID_091FC92A_99C1_56CD_77D7_E72BA09F6857'}
	(* Computes the natural exponent of each pixel value. *)
	FUNCTION F_VN_ElementwiseExp : HRESULT
	VAR_INPUT
		ipSrcImage	:	ITcVnImage;	(* Source image (REAL or LREAL) *)
		ipDestImage	:	REFERENCE TO ITcVnImage;	(* Destination image (Same type and size as ipSrcImage, an appropriate image will be created if required.) *)
		hrPrev	:	HRESULT;	(* HRESULT indicating the result of previous operations (If SUCCEEDED(hrPrev) equals false, no operation is executed.) *)
	END_VAR

END_FUNCTION

// Functions/Algebraic Image Operations/F_VN_ElementwiseLog

	{attribute 'TcIecLibraryType'}
	{attribute 'external_name' := 'F_VN_ElementwiseLog_GUID_11C8D313_3B6E_50D3_4E63_2A41DC742A1E'}
	(* Computes the natural logarithm of each pixel value. *)
	FUNCTION F_VN_ElementwiseLog : HRESULT
	VAR_INPUT
		ipSrcImage	:	ITcVnImage;	(* Source image (REAL or LREAL) *)
		ipDestImage	:	REFERENCE TO ITcVnImage;	(* Destination image (Same type and size as ipSrcImage, an appropriate image will be created if required.) *)
		hrPrev	:	HRESULT;	(* HRESULT indicating the result of previous operations (If SUCCEEDED(hrPrev) equals false, no operation is executed.) *)
	END_VAR

END_FUNCTION

// Functions/Algebraic Image Operations/F_VN_MaxImage

	{attribute 'TcIecLibraryType'}
	{attribute 'external_name' := 'F_VN_MaxImage_GUID_71815673_6575_5427_4DCA_28682DA3447B'}
	(* Element-wise maximum of two images. *)
	FUNCTION F_VN_MaxImage : HRESULT
	VAR_INPUT
		ipSrcImage1	:	ITcVnImage;	(* First source image *)
		ipSrcImage2	:	ITcVnImage;	(* Second source image *)
		ipDestImage	:	REFERENCE TO ITcVnImage;	(* Destination image (An appropriate destination image will be created if required.) *)
		hrPrev	:	HRESULT;	(* HRESULT indicating the result of previous operations (If SUCCEEDED(hrPrev) equals false, no operation is executed.) *)
	END_VAR

END_FUNCTION

// Functions/Algebraic Image Operations/F_VN_MaxImageExp

	{attribute 'TcIecLibraryType'}
	{attribute 'external_name' := 'F_VN_MaxImageExp_GUID_7FCCC36E_AF44_5FE5_6A0F_8639C5F774A3'}
	(* Element-wise maximum of two images. (expert function) *)
	FUNCTION F_VN_MaxImageExp : HRESULT
	VAR_INPUT
		ipSrcImage1	:	ITcVnImage;	(* First source image *)
		ipSrcImage2	:	ITcVnImage;	(* Second source image *)
		ipDestImage	:	REFERENCE TO ITcVnImage;	(* Destination image (An appropriate destination image will be created if required.) *)
		ipMask	:	ITcVnImage;	(* Mask of type USINT *)
		hrPrev	:	HRESULT;	(* HRESULT indicating the result of previous operations (If SUCCEEDED(hrPrev) equals false, no operation is executed.) *)
	END_VAR

END_FUNCTION

// Functions/Algebraic Image Operations/F_VN_MaxImageWithScalar

	{attribute 'TcIecLibraryType'}
	{attribute 'external_name' := 'F_VN_MaxImageWithScalar_GUID_24412284_C75F_5852_7B4D_52C6CCD7D8AF'}
	(* Element-wise maximum of image and scalar value. *)
	FUNCTION F_VN_MaxImageWithScalar : HRESULT
	VAR_INPUT
		fScalar	:	LREAL;	(* Scalar value *)
		ipSrcImage	:	ITcVnImage;	(* Source image *)
		ipDestImage	:	REFERENCE TO ITcVnImage;	(* Destination image (An appropriate destination image will be created if required.) *)
		hrPrev	:	HRESULT;	(* HRESULT indicating the result of previous operations (If SUCCEEDED(hrPrev) equals false, no operation is executed.) *)
	END_VAR

END_FUNCTION

// Functions/Algebraic Image Operations/F_VN_MaxImageWithScalarExp

	{attribute 'TcIecLibraryType'}
	{attribute 'external_name' := 'F_VN_MaxImageWithScalarExp_GUID_54728949_28DD_5692_7D25_DBD37150313D'}
	(* Element-wise maximum of image and scalar value. (expert function) *)
	FUNCTION F_VN_MaxImageWithScalarExp : HRESULT
	VAR_INPUT
		fScalar	:	LREAL;	(* Scalar value *)
		ipSrcImage	:	ITcVnImage;	(* Source image *)
		ipDestImage	:	REFERENCE TO ITcVnImage;	(* Destination image (An appropriate destination image will be created if required.) *)
		ipMask	:	ITcVnImage;	(* Mask of type USINT *)
		hrPrev	:	HRESULT;	(* HRESULT indicating the result of previous operations (If SUCCEEDED(hrPrev) equals false, no operation is executed.) *)
	END_VAR

END_FUNCTION

// Functions/Algebraic Image Operations/F_VN_MaxImageWithVector

	{attribute 'TcIecLibraryType'}
	{attribute 'external_name' := 'F_VN_MaxImageWithVector_GUID_C630AD8B_1483_5F10_63EF_E516771892CC'}
	(* Element-wise maximum of image and vector (1 element for each image channel). *)
	FUNCTION F_VN_MaxImageWithVector : HRESULT
	VAR_INPUT
		aVector	:	REFERENCE TO TcVnVector4_LREAL;	(* 4-element vector (1 element for each image channel. If the image has less channels, the further vector elements are ignored.) *)
		ipSrcImage	:	ITcVnImage;	(* Source image *)
		ipDestImage	:	REFERENCE TO ITcVnImage;	(* Destination image (An appropriate destination image will be created if required.) *)
		hrPrev	:	HRESULT;	(* HRESULT indicating the result of previous operations (If SUCCEEDED(hrPrev) equals false, no operation is executed.) *)
	END_VAR

END_FUNCTION

// Functions/Algebraic Image Operations/F_VN_MaxImageWithVectorExp

	{attribute 'TcIecLibraryType'}
	{attribute 'external_name' := 'F_VN_MaxImageWithVectorExp_GUID_D6DDCE49_8BC3_557A_629B_29E84C8EA503'}
	(* Element-wise maximum of image and vector (1 element for each image channel). (expert function) *)
	FUNCTION F_VN_MaxImageWithVectorExp : HRESULT
	VAR_INPUT
		aVector	:	REFERENCE TO TcVnVector4_LREAL;	(* 4-element vector (1 element for each image channel. If the image has less channels, the further vector elements are ignored.) *)
		ipSrcImage	:	ITcVnImage;	(* Source image *)
		ipDestImage	:	REFERENCE TO ITcVnImage;	(* Destination image (An appropriate destination image will be created if required.) *)
		ipMask	:	ITcVnImage;	(* Mask of type USINT *)
		hrPrev	:	HRESULT;	(* HRESULT indicating the result of previous operations (If SUCCEEDED(hrPrev) equals false, no operation is executed.) *)
	END_VAR

END_FUNCTION

// Functions/Algebraic Image Operations/F_VN_MinImage

	{attribute 'TcIecLibraryType'}
	{attribute 'external_name' := 'F_VN_MinImage_GUID_11197D17_38AE_5A63_668B_09D083426B9C'}
	(* Element-wise minimum of two images. *)
	FUNCTION F_VN_MinImage : HRESULT
	VAR_INPUT
		ipSrcImage1	:	ITcVnImage;	(* First source image *)
		ipSrcImage2	:	ITcVnImage;	(* Second source image *)
		ipDestImage	:	REFERENCE TO ITcVnImage;	(* Destination image (An appropriate destination image will be created if required.) *)
		hrPrev	:	HRESULT;	(* HRESULT indicating the result of previous operations (If SUCCEEDED(hrPrev) equals false, no operation is executed.) *)
	END_VAR

END_FUNCTION

// Functions/Algebraic Image Operations/F_VN_MinImageExp

	{attribute 'TcIecLibraryType'}
	{attribute 'external_name' := 'F_VN_MinImageExp_GUID_F5D8A639_467E_5F3F_53C2_77B444FDBD34'}
	(* Element-wise minimum of two images. (expert function) *)
	FUNCTION F_VN_MinImageExp : HRESULT
	VAR_INPUT
		ipSrcImage1	:	ITcVnImage;	(* First source image *)
		ipSrcImage2	:	ITcVnImage;	(* Second source image *)
		ipDestImage	:	REFERENCE TO ITcVnImage;	(* Destination image (An appropriate destination image will be created if required.) *)
		ipMask	:	ITcVnImage;	(* Mask of type USINT *)
		hrPrev	:	HRESULT;	(* HRESULT indicating the result of previous operations (If SUCCEEDED(hrPrev) equals false, no operation is executed.) *)
	END_VAR

END_FUNCTION

// Functions/Algebraic Image Operations/F_VN_MinImageWithScalar

	{attribute 'TcIecLibraryType'}
	{attribute 'external_name' := 'F_VN_MinImageWithScalar_GUID_FCC06F57_8AA1_5C7E_4E60_1269E61A6489'}
	(* Element-wise minimum of image and scalar value. *)
	FUNCTION F_VN_MinImageWithScalar : HRESULT
	VAR_INPUT
		fScalar	:	LREAL;	(* Scalar value *)
		ipSrcImage	:	ITcVnImage;	(* Source image *)
		ipDestImage	:	REFERENCE TO ITcVnImage;	(* Destination image (An appropriate destination image will be created if required.) *)
		hrPrev	:	HRESULT;	(* HRESULT indicating the result of previous operations (If SUCCEEDED(hrPrev) equals false, no operation is executed.) *)
	END_VAR

END_FUNCTION

// Functions/Algebraic Image Operations/F_VN_MinImageWithScalarExp

	{attribute 'TcIecLibraryType'}
	{attribute 'external_name' := 'F_VN_MinImageWithScalarExp_GUID_39D76814_023C_5052_4FCA_954D873E0FCC'}
	(* Element-wise minimum of image and scalar value. (expert function) *)
	FUNCTION F_VN_MinImageWithScalarExp : HRESULT
	VAR_INPUT
		fScalar	:	LREAL;	(* Scalar value *)
		ipSrcImage	:	ITcVnImage;	(* Source image *)
		ipDestImage	:	REFERENCE TO ITcVnImage;	(* Destination image (An appropriate destination image will be created if required.) *)
		ipMask	:	ITcVnImage;	(* Mask of type USINT *)
		hrPrev	:	HRESULT;	(* HRESULT indicating the result of previous operations (If SUCCEEDED(hrPrev) equals false, no operation is executed.) *)
	END_VAR

END_FUNCTION

// Functions/Algebraic Image Operations/F_VN_MinImageWithVector

	{attribute 'TcIecLibraryType'}
	{attribute 'external_name' := 'F_VN_MinImageWithVector_GUID_DD0D2C46_9907_59CB_583F_E99F692ABF53'}
	(* Element-wise minimum of image and vector (1 element for each image channel). *)
	FUNCTION F_VN_MinImageWithVector : HRESULT
	VAR_INPUT
		aVector	:	REFERENCE TO TcVnVector4_LREAL;	(* 4-element vector (1 element for each image channel. If the image has less channels, the further vector elements are ignored.) *)
		ipSrcImage	:	ITcVnImage;	(* Source image *)
		ipDestImage	:	REFERENCE TO ITcVnImage;	(* Destination image (An appropriate destination image will be created if required.) *)
		hrPrev	:	HRESULT;	(* HRESULT indicating the result of previous operations (If SUCCEEDED(hrPrev) equals false, no operation is executed.) *)
	END_VAR

END_FUNCTION

// Functions/Algebraic Image Operations/F_VN_MinImageWithVectorExp

	{attribute 'TcIecLibraryType'}
	{attribute 'external_name' := 'F_VN_MinImageWithVectorExp_GUID_7262ABCF_1ED7_55B1_6C64_6E982310B046'}
	(* Element-wise minimum of image and vector (1 element for each image channel). (expert function) *)
	FUNCTION F_VN_MinImageWithVectorExp : HRESULT
	VAR_INPUT
		aVector	:	REFERENCE TO TcVnVector4_LREAL;	(* 4-element vector (1 element for each image channel. If the image has less channels, the further vector elements are ignored.) *)
		ipSrcImage	:	ITcVnImage;	(* Source image *)
		ipDestImage	:	REFERENCE TO ITcVnImage;	(* Destination image (An appropriate destination image will be created if required.) *)
		ipMask	:	ITcVnImage;	(* Mask of type USINT *)
		hrPrev	:	HRESULT;	(* HRESULT indicating the result of previous operations (If SUCCEEDED(hrPrev) equals false, no operation is executed.) *)
	END_VAR

END_FUNCTION

// Functions/Algebraic Image Operations/F_VN_MultiplyImages

